°C 		v 				h 			u 		s 			cp 		Y 		L		n		s	
-20		1,006580	
0 		1,000160 		0,06 		-0,04 	-0,0001 	4,228 	-0,080 	561,0 	1792 	75,65
4		1,000028
5 		1,0000 		21,1 		21,0 	0,076 		4,200 	0,011 	570,6 	1518 	74,95
10 		1,0003 		42,1 		42,0 	0,151 		4,188 	0,087 	580,0 	1306 	74,22
15 		1,0009 		63,0 		62,9 	0,224 		4,184 	0,152 	589,4 	1137 	73,49
20 		1,001797 		83,9 		83,8 	0,296 		4,183 	0,209 	598,4 	1001 	72,74
25 		1,0029 		104,8 		104,7 	0,367 		4,183 	0,259 	607,2 	890,4 	71,98
30 		1,0044 		125,8 		125,7 	0,437 		4,183 	0,305 	615,5 	797,7 	71,20
35 		1,0060 		146,7 		146,6 	0,505 		4,183 	0,347 	623,3 	719,6 	70,41
40 		1,007842 		167,58 	167,5 	0,572 		4,182 	0,386 	630,6 	653,3 	69,60
45 		1,0099 		188,5 		188,4 	0,638 		4,182 	0,423 	637,3 	596,3 	68,78
50 		1,0121 		209,4 		209,3 	0,704 		4,181 	0,457 	643,6 	547,1 	67,95
60 		1,017089 		251,2 		251,1 	0,831 		4,183 	0,522 	654,4 	466,6 	66,24
70 		1,0227 		293,1 		293,0 	0,955 		4,187 	0,583 	663,1 	404,1 	64,49
80 		1,029027 		335,0 		334,9 	1,075 		4,194 	0,640 	670,0 	354,5 	62,68
90 		1,0359 		377,0 		376,9 	1,193 		4,204 	0,696 	675,3 	314,6 	60,82
99,63 	1,0431 		417,5 		417,4 	1,303 		4,217 	0,748 	679,0 	283,0 	58,99
100	1,043453		419,1

Stoffdaten von Wasser Quelle Wickipedia

Wasser hat unter Normaldruck seine größte Dichte von 1000 Kilogramm pro Kubikmeter bei 3,98 °C und zeigt damit eine Dichteanomalie. 
Diese besteht darin, dass sich Wasser unterhalb von 3,98 °C bei weiterer Temperaturverringerung, auch beim Wechsel zum festen 
Aggregatzustand, wieder ausdehnt, was man nur von wenigen Stoffen kennt. Die derzeit genauesten publizierten Werte für die maximale 
Dichte liegen bei (999,974950 ± 0,00084) kg/m³ und bei (3,983 ± 0,00067) °C für die Temperatur, bei der dieser Wert erreicht wird. 
Die Werte stellen einen Mittelwert der von verschiedenen physikalischen Instituten veröffentlichten Zahlen dar (Stand 2001).

Die Berechnung der Dichte von luftfreiem Wasser DLF in Abhängigkeit von der Temperatur T ([T] = °C) kann mit Hilfe der folgenden 
Virialgleichung erfolgen:
: \frac{D_{\rm LF}}{\rm g/l} = \frac{a_0 + a_1 T + a_2 T^2 + a_3 T^3 + a_4 T^4 + a_5 T^5}{1 + b T}.
mit den Koeffizienten: a0 = 999,83952; a1 = 16,952577 (°C)-1; a2 = -7,9905127·10-3 (°C)-2; a3 = -4,6241757·10-5 (°C)-3; 
a4 = 1,0584601·10-7 (°C)-4; a5 = -2,8103006·10-10 (°C)-5 und b = 0,0168872. 
Für die Berechnung der Dichte von luftgesättigtem Wasser korrigiert man den Wert nach 
DLG/(g/l) = DLF/(g/l) - 0,004612 + 0,000106 (°C)-1·T. (Quelle: PTB-Mitteilungen 100/3-90)

*)
END_FUNCTION

(* POU Mathematical/functions/LINEAR_INT, ST *)
FUNCTION LINEAR_INT : REAL
VAR_INPUT
	X : REAL;
	XY : ARRAY[1..20,0..1] OF REAL;
	Pts : INT;
END_VAR
VAR
	i : INT;
END_VAR

(*
	version 1.1	27 dec 2007
	programmer 	oscat
	tested BY		oscat

LINEAR_INT calculates an output based on a linear interpolation of up to 20 coordinates given in an array
the input coordinates have to start at the lowest array position and must be sorted ba ascending X values.

*)
(*make sure n is bound within the array size *)
pts := MIN(pts,20);

(* calculate the linear segement interpolation *)
i := 2;
(* search for segment and calculate output
	below and above the defined segments we interpolate the last segment *)
WHILE (i < pts) AND (XY[i,0] < X) DO
	i := i + 1;
END_WHILE;

(* calculate the output value on the corresponding segment coordinates *)
LINEAR_INT := ((XY[i,1] - XY[i-1,1]) * X - XY[i,1] * XY[i-1,0] + XY[i-1,1] * XY[i,0]) / (XY[i,0] - XY[i-1,0]);

(* revision history
hm	7. oct 2007		rev 1.0
	original version

hm	27 dec 2007		rev 1.1
	changed code for better performance
*)
END_FUNCTION

(* POU Building/HLK/Heat_temp, ST *)
FUNCTION_BLOCK Heat_temp
VAR_INPUT
	T_ext : REAL;
	Offset : REAL;
	t_req : REAL;
END_VAR
VAR_INPUT CONSTANT
	TY_max : REAL := 70;
	TY_min : REAL := 20;
	T_int : REAL := 20;
	TY_config : REAL := 50;
	T_ext_config : REAL := -15;
	C : REAL := 1.33;
END_VAR
VAR_OUTPUT
	Ty : REAL;
END_VAR
VAR
END_VAR

(*
version 1.0	27 jan 2007
programmer 	hugo
tested by		tobias

Heat_Temp calculates a heat characteristic based on the formula: tv=ti+(tvmax-ti)*((ti-tau)/(ti-taumin))^(1/n)
while
tv necessary heating temperature.
ti internal room temperature (20°C)
tau current external temperature
external temperature to determine characteristics
C exponent for heating system (normally 1,33 or 1,1 for floor heating)

The two additional inputs TY_min and TY_max set limits for the output TY, while an offset inputs allows to rise or lower the room temperature.

*)
IF t_ext > t_int + Offset THEN
	ty := t_int + offset;
ELSE
Ty := T_int - offset + (TY_config - T_int) * EXPT((T_int - offset - T_ext) / (T_int - offset - T_ext_config),1 / C);
END_IF;
IF t_req > ty THEN ty := t_req; END_IF;
ty := LIMIT(TY_min, ty, TY_max);



(*

tv=ti+(tvmax-ti)*((ti-tau)/(ti-taumin))^(1/n)

tv aktuelle Vorlauftemp.
ti Raumtemperatur innen (20°C)
tau aktuelle Außentemperatur
taumin minimale Außentemperatur -12°C oder -15°C
n Heizkörperexponent (meistens 1,33)
Fußbodenheizung = 1,1
Wandheizung 1,3

Normen z. B. DIN 4703, DIN 4725 oder die Literatur, z. B Recknagel Abschnitt 1.3.5.

*)
END_FUNCTION_BLOCK

(* POU Building/HLK/legionella, ST *)
FUNCTION_BLOCK legionella
VAR_INPUT
	manual : BOOL;
	temp_boiler : REAL;
	temp_return : REAL := 100;
	DT_in: DT;
	rst : BOOL;
END_VAR
VAR_INPUT CONSTANT
	T_start: TOD := tod#03:00:00;
	day : INT := 7;
	temp_set : REAL := 70;
	temp_offset : REAL := 10;
	temp_hys : REAL := 5;
	t_max_heat: TIME := t#10m;
	t_max_ret : TIME := t#10m;
	tp_0: TIME := t#5m;
	tp_1: TIME := t#5m;
	tp_2: TIME := t#5m;
	tp_3: TIME := t#5m;
	tp_4: TIME := t#5m;
	tp_5: TIME := t#5m;
	tp_6: TIME := t#5m;
	tp_7: TIME := t#5m;
END_VAR
VAR_OUTPUT
	Heat : BOOL;
	pump : BOOL;
	valve0 : BOOL;
	valve1 : BOOL;
	valve2 : BOOL;
	valve3 : BOOL;
	valve4 : BOOL;
	valve5 : BOOL;
	valve6 : BOOL;
	valve7 : BOOL;
	run: BOOL;
	Status : BYTE;
END_VAR
VAR
	X1: timer_1;
	x2: sequence_8;
	x3: hyst_1;
	init: BOOL;
END_VAR

(*
version 1.1	17. jan 2007
programmer 	oscat
tested by		hans

Legionella is a complete sequencer for up to 8 hot water lines that need to be sterilzed periodically.
legionella needs a DT input with the appropriate time, usually gererated by the rtc of the system. for system independence this time is connected externally.
T_start is the time when sterilazation should be started and day is the day_of_week when it should be performed (1=Monday and 7=sunday).
so sterilazation is autioimatically performed once a week at a specified time.
temp_set and temp_hys and temp_offset specify the boiler temperatur nedded for sterilization. as a defaut Temp_set is set to 70 deg C and Temp_hys is set to 5 deg C and temp_offset is 10 deg C.
a temp boiler input reads the boiler temperature of the hot water tank.
after a start pulse is gererated by the weekly timer or a manual test input the sequence is started:
1. the boiler is heated to temp_set + temp_offset + temp_hys = 85 deg C unless chaged at setup.
	the heat output is turned on and tells the heater to turn heating on. if the temp is not reached for a time of t_max_heat (10 min) the error output is set and the sequence is stopped.
2. after the specified temperature is reached, the output valve0 and pump is turned on and starts sterilization of line0 until temp_return has reached temp_set and continues to sterilize for a time of tp_0 (5 min default).
	if tmep_set is not reached at the temp_return_input then the error output is set and the sequence will be stopped.
	if there is no temp sensor for temp_return (the temperature at the return point for the circulation pump pls set this imput to a value greater then temp_set (by default use 100 deg C).
	in this case sterilization is performed for the default times without monitoring the return temp.
3. this sequence is repeated for up to valves.

connection scheme:

temp_boiler:	input oif the boiler temperature sensor.
temp_hys:		config value for the heater hysteresis, preset to 5 deg C.
temp_offset:	config value for the heater temp_offset against temp_set, preset to 10 deg C.
temp_set:		config value for the specified sterilization temperature, preset to 70 deg C.
temp_return:	input of the circulation return line temperature sensor, if not availabe set this value to 100 deg C.
manual:		manual input to start the sterilization by hand for diagnostic purposes, rising edge active, leave low for automatic operation.
DT_in:			date,time input supplied by a external real time clock.
T_start:		time of day when the sterilization should be started.
day:			config value for day of week when the process should be started, preset to sunday.
t_max_hest:	tmax time to be needed for the heater to heat the hot water tank to the specified value, preset to 10 min.

*)
(* startup initialization *)
IF NOT init THEN
	init := TRUE;
	X1.start_day := day;
	X1.start_time := T_start;
	X3.low := Temp_offset + temp_set;
	X3.high := Temp_hys + X3.low;
	X2.wait0 := T_max_heat;
	X2.delay0 := TP_0;
	X2.delay1 := TP_1;
	X2.delay2 := TP_2;
	X2.delay3 := TP_3;
	X2.delay4 := TP_4;
	X2.delay5 := TP_5;
	X2.delay6 := TP_6;
	X2.delay7 := TP_7;
	X2.wait1 := T_max_ret;
	X2.wait2 := T_max_ret;
	X2.wait3 := T_max_ret;
	X2.wait4 := T_max_ret;
	X2.wait5 := T_max_ret;
	X2.wait6 := T_max_ret;
	X2.wait7 := T_max_ret;
	X2();
END_IF;

(* oerational code *)
X1(DT_in := DT_in);
IF X1.Q OR manual OR x2.run THEN
	X3(in := temp_boiler);
	X2.in0 := X3.Q OR x3.win;
	X2.in1 := temp_return >= temp_set;
	X2.in2 := x2.in1;
	X2.in3 := x2.in1;
	X2.in4 := x2.in1;
	X2.in5 := x2.in1;
	X2.in6 := x2.in1;
	X2.in7 := x2.in1;
	X2.rst := rst;
	X2(start := X1.Q OR manual);
	run := x2.run;
	pump := x2.any;
	Heat := NOT X3.Q AND x2.run;
	valve0 := X2.Q0;
	valve1 := X2.Q1;
	valve2 := X2.Q2;
	valve3 := X2.Q3;
	valve4 := X2.Q4;
	valve5 := X2.Q5;
	valve6 := X2.Q6;
	valve7 := X2.Q7;
	pump := X2.any;
	status := X2.status;
ELSE;
	X2(start :=0);
	status := x2.status;
END_IF;

(* revision history

hm 17.jan 2007	rev 1.1
	rewritten to st for higher performance
	changes eeror output to esr compatible status output
*)
END_FUNCTION_BLOCK

(* POU Logic/generators/sequence_8, ST *)
FUNCTION_BLOCK sequence_8
VAR_INPUT
	in0 : BOOL := TRUE;
	in1 : BOOL := TRUE;
	in2 : BOOL := TRUE;
	in3 : BOOL := TRUE;
	in4 : BOOL := TRUE;
	in5 : BOOL := TRUE;
	in6 : BOOL := TRUE;
	in7 : BOOL := TRUE;
	start : BOOL;
	rst : BOOL;
	wait0 : TIME := t#0s;
	delay0 : TIME := t#0s;
	wait1 : TIME := t#0s;
	delay1 : TIME := t#0s;
	wait2 : TIME := t#0s;
	delay2 : TIME := t#0s;
	wait3 : TIME := t#0s;
	delay3 : TIME := t#0s;
	wait4 : TIME := t#0s;
	delay4 : TIME := t#0s;
	wait5 : TIME := t#0s;
	delay5 : TIME := t#0s;
	wait6 : TIME := t#0s;
	delay6 : TIME := t#0s;
	wait7 : TIME := t#0s;
	delay7 : TIME := t#0s;
END_VAR
VAR_INPUT CONSTANT
	stop_on_error : BOOL := FALSE;
END_VAR
VAR_OUTPUT
	Q0 : BOOL;
	Q1 : BOOL;
	Q2 : BOOL;
	Q3 : BOOL;
	Q4 : BOOL;
	Q5 : BOOL;
	Q6 : BOOL;
	Q7 : BOOL;
	any : BOOL;
	run: BOOL;
	step : INT := -1;
	status : BYTE;
END_VAR
VAR
	last : TIME;
	edge : BOOL;
	tx: TIME;
	init: BOOL;
END_VAR

(*
version 1.4	17 sep 2007
programmer 	oscat
tested by		hans

sequence_8 enables run when a low to high transition is present on start.
a low to high transition on start will restart the sequencer at any time while a rst will hold the sequencer in reset while true.
after run is enabled with a rising edge on start the sequencer waits for wait0 on in0 to enable q0 which stays on for delay0.
the next cycle starts with wait1, continues with delay 1 and so on...
if an edge is not detected during the wait period, the sequencer will then display the error number on the status output.
The status numbers are 1 .. 8 for erros in step 0..7.
after the last step that sets q7, the sequencer leaves q7 on for delay7 and then resets to the initial state.
a step output will indicate the current step of the sequencer and will also be present with a fault condition.
after the first output is turened on the sequencer switches from q0 to q1 and so on, at any time there is only one output enabled.
if an input signal is not detected during a wait period, the sequencer will display the error number ( 1 for in0, 2 for in1 .... ).
when an error is present and the config variable stop_on_error is set then the sequencer will stop. otherwise it will continue.
The status output will also display 110 for waiting and 111 sequece running.

*)
(* read sps timer *)
tx := DWORD_TO_TIME(T_PLC_MS());

(* initialize on startup *)
IF NOT init THEN
	last := tx;
	init := TRUE;
	status := 110;
END_IF;

(* asynchronous reset *)
IF rst THEN
	step := -1;
	Q0 := 0;
	Q1 := 0;
	Q2 := 0;
	Q3 := 0;
	Q4 := 0;
	Q5 := 0;
	Q6 := 0;
	Q7 := 0;
	status := 110;
	run := 0;

(* edge on start input restarts the sequencer *)
ELSIF start AND NOT edge THEN
	step := 0;
	last := tx;
	status := 111;
	Q0 := 0;
	Q1 := 0;
	Q2 := 0;
	Q3 := 0;
	Q4 := 0;
	Q5 := 0;
	Q6 := 0;
	Q7 := 0;
	run := 1;
END_IF;
edge := start;

(* check if stop on error is necessary *)
IF status > 0 AND status < 100 AND stop_on_error THEN RETURN; END_IF;

(* sequence is running *)
IF run AND step = 0 THEN
	IF NOT q0 AND in0 AND tx - last <= wait0 THEN
		Q0 := TRUE;
		last := tx;
	ELSIF NOT q0 AND tx - last > wait0 THEN
		status := 1;
		run := FALSE;
	ELSIF q0 AND tx - last >= delay0 THEN
		step := 1;
		last := tx;
	END_IF;
END_IF;
IF run AND step = 1 THEN
	IF NOT q1 AND in1 AND tx - last <= wait1 THEN
		Q0 := FALSE;
		Q1 := TRUE;
		last := tx;
	ELSIF NOT q1 AND Tx - last > wait1 THEN
		status := 2;
		q0 := FALSE;
		run := FALSE;
	ELSIF q1 AND tx - last >= delay1 THEN
		step := 2;
		last := tx;
	END_IF;
END_IF;
IF run AND step = 2 THEN
	IF NOT q2 AND in2 AND tx - last <= wait2 THEN
		Q1 := FALSE;
		Q2 := TRUE;
		last := tx;
	ELSIF NOT q2 AND Tx - last > wait2 THEN
		status := 3;
		q1 := FALSE;
		run := FALSE;
	ELSIF q2 AND tx - last >= delay2 THEN
		step := 3;
		last := tx;
	END_IF;
END_IF;
IF run AND step = 3 THEN
	IF NOT q3 AND in3 AND tx - last <= wait3 THEN
		Q2 := FALSE;
		Q3 := TRUE;
		last := tx;
	ELSIF NOT q3 AND Tx - last > wait3 THEN
		status := 4;
		q2 := FALSE;
		run := FALSE;
	ELSIF q3 AND tx - last >= delay3 THEN
		step := 4;
		last := tx;
	END_IF;
END_IF;
IF run AND step = 4 THEN
	IF NOT q4 AND in4 AND tx - last <= wait4 THEN
		Q3 := FALSE;
		Q4 := TRUE;
		last := tx;
	ELSIF NOT q4 AND Tx - last > wait4 THEN
		status := 5;
		q3 := FALSE;
		run := FALSE;
	ELSIF q4 AND tx - last >= delay4 THEN
		step := 5;
		last := tx;
	END_IF;
END_IF;
IF run AND step = 5 THEN
	IF NOT q5 AND in5 AND tx - last <= wait5 THEN
		Q4 := FALSE;
		Q5 := TRUE;
		last := tx;
	ELSIF NOT q5 AND Tx - last > wait5 THEN
		status := 6;
		q4 := FALSE;
		run := FALSE;
	ELSIF q5 AND tx - last >= delay5 THEN
		step := 6;
		last := tx;
	END_IF;
END_IF;
IF run AND step = 6 THEN
	IF NOT q6 AND in6 AND tx - last <= wait6 THEN
		Q5 := FALSE;
		Q6 := TRUE;
		last := tx;
	ELSIF NOT q6 AND Tx - last > wait6 THEN
		status := 7;
		q5 := FALSE;
		run := FALSE;
	ELSIF q6 AND tx - last >= delay6 THEN
		step := 7;
		last := tx;
	END_IF;
END_IF;
IF run AND step = 7 THEN
	IF NOT q7 AND in7 AND tx - last <= wait7 THEN
		Q6 := FALSE;
		Q7 := TRUE;
		last := tx;
	ELSIF NOT q7 AND Tx - last > wait7 THEN
		status := 8;
		q6 := FALSE;
		run := FALSE;
	ELSIF q7 AND tx - last >= delay7 THEN
		step := -1;
		Q7 := FALSE;
		Run := FALSE;
		status := 110;
	END_IF;
END_IF;
any := q0 OR q1 OR q2 OR q3 OR q4 OR q5 OR q6 OR q7;

(*
hm 1.10.06		rev 1.1
	corrected delay logic to be after event and not before
	added any output

hm 1.12.06		rev 1.2
	corrected failure in sequence logic.
	added init at startup to prevent from initial statuss after start.

hm 17.1.2007		rev 1.3
	changed output fault to status for better compatibility with other modules (ESR)
	added stop on error functionality and setup variable
	default for inputs in0..7 is true.
	renames variable state to step

hm	17.sep 2007		rev 1.4
	replaced time() with T_PLC_MS() for compatibility reasons

*)
END_FUNCTION_BLOCK

(* POU Engineering/control/hyst_1, ST *)
FUNCTION_BLOCK hyst_1
VAR_INPUT
	In : REAL;
	high : REAL;
	low : REAL;
END_VAR
VAR_OUTPUT
	Q : BOOL := 0;
	win : BOOL := 0;
END_VAR
VAR
END_VAR

(*
	version 1.0	4 aug 2006
	programmer 	hugo
	tested BY		tobias

this hysteresis function switches the output high if the input signal reaches obove high and will switch to low when the input falls back below low value.
a separate output mid is set if the input stays between low and high value.

*)
IF Q THEN
	IF in < low THEN q := FALSE; END_IF;
ELSE
	IF in > high THEN q := TRUE; END_IF;
END_IF;
win := in > low AND in < high;
END_FUNCTION_BLOCK

(* POU Building/HLK/temp_ext, ST *)
FUNCTION_BLOCK temp_ext
VAR_INPUT
	t_ext1 : REAL;
	t_ext2 : REAL;
	t_ext3 : REAL;
	t_ext_config : BYTE := 0;
	dt_in : DT;
END_VAR
VAR_INPUT CONSTANT
	t_ext_min : REAL := -40;
	t_ext_max : REAL := 60;
	t_ext_default : REAL := -10;
	heat_period_start : DATE := D#1970-9-1;
	heat_period_stop : DATE := D#1970-4-30;
	cool_period_start : DATE := D#1970-4-1;
	cool_period_stop : DATE := D#1970-9-30;
	heat_start_temp_day : REAL := 15;
	heat_start_temp_night : REAL := 10;
	heat_stop_temp : REAL := 18;
	cool_start_temp_day : REAL := 26;
	cool_start_temp_night : REAL := 26;
	cool_stop_temp : REAL := 24;
	start_day : TOD := tod#09:00;
	start_night : TOD := tod#21:00;
	cycle_time : TIME := t#10m;
END_VAR
VAR_OUTPUT
	t_ext : REAL;
	heat : BOOL;
	cool : BOOL;
END_VAR
VAR
	tx: TIME;
	last_run: TIME;
	init: BOOL;
	cool_start: DATE;
	cool_stop: DATE;
	heat_start: DATE;
	heat_stop: DATE;
	xdate: DATE;
	day: BOOL;
END_VAR


(*
version 1.1	15 sep 2007
programmer 	hugo
tested by		tobias

temp_ext measures and processes ext temperature and decides if heating or cooling is needed.

 the measurement of t_ext has 3 inputs which can be configured in different ways:
	t_ext_config = 0 means the ext temp is the avg of the 3 external temperatures, this mode is the default mode.
	t_ext_config = 1 means t_ext1 is used.
	t_ext_config = 2 means t_ext1 is used.
	t_ext_config = 3 means t_ext1 is used.
	t_ext_config = 4 means t_ext_default is used.
	t_ext_config = 5 means the lowest of the 3 external temperatures is used.
	t_ext_config = 6 means the higest externnal temperature is used.
	t_ext_config = 7 means the midlle external temperature is used, if there are only two working, the lowest is used.
	in any config mode, an external temperature higher then t_ext_max or lower then t_ext_min is ignored to prevent from temperatures caused by broken sensors or wires.
	if no external temperature is available, a default value (t_ext_default) is used.
	if you have only one external sensor, connect the 3 inputs to the same sensor, or select the right input with t_ext_config.

heating or cooling is enabled during heating / cooling period when the day or night start temperature is reached for at least the specified delay time and will be disabled after the stop temperature is reached. 
t_ext output can be used by other modules to determine the correct system temperature for heating or cooling.

*)
IF NOT init THEN
	init := TRUE;
	heat_start := set_Date(1972,month(heat_period_start),day_of_month(heat_period_start));
	heat_stop := set_Date(1972,month(heat_period_stop),day_of_month(heat_period_stop));
	cool_start := set_Date(1972,month(cool_period_start),day_of_month(cool_period_start));
	cool_stop := set_Date(1972,month(cool_period_stop),day_of_month(cool_period_stop));
END_IF;

(* read system time *)
tx := DWORD_TO_TIME(T_PLC_MS());

(* for efficiency exit isf this program has been executed less then 1min ago *)
IF tx - last_run < cycle_time THEN RETURN; END_IF;

(* calculate frequently used variables *)
xdate := set_Date(1972,month(DT_TO_DATE(dt_in)),day_of_month(DT_TO_DATE(dt_in)));
day := DT_TO_TOD(dt_in) >= start_day AND  DT_TO_TOD(dt_in) < start_night;

(* read the correct external temperature depending on the t_ext_config setting *)
t_ext := multi_in(t_ext1, t_ext2, t_ext3, t_ext_default, t_ext_min, t_ext_max, t_ext_config);

(* dtermine heating *)
IF (heat_start <= heat_stop AND xdate >= heat_start AND xdate <= heat_stop) OR (heat_start > heat_stop AND (xdate >= heat_start OR xdate <= heat_stop)) THEN
	(* heating period id true check for temperature *)
	IF day AND t_ext <= heat_start_temp_day THEN
		heat := TRUE;
	ELSIF NOT day AND t_ext <= heat_start_temp_night THEN
		heat := TRUE;
	ELSIF t_ext >= heat_stop_temp THEN
		heat := FALSE;
	END_IF;
ELSE
	heat := FALSE;
END_IF;

(* dtermine cooling *)
IF (cool_start <= cool_stop AND xdate >= cool_start AND xdate <= cool_stop) OR (cool_start > cool_stop AND (xdate >= cool_start OR xdate <= cool_stop)) THEN
	(* cooling period is true check for temperature *)
	IF day AND t_ext >= cool_start_temp_day THEN
		cool := TRUE;
	ELSIF NOT day AND t_ext >= cool_start_temp_night THEN
		cool := TRUE;
	ELSIF t_ext <= cool_stop_temp THEN
		cool := FALSE;
	END_IF;
ELSE
	cool := FALSE;
END_IF;

last_run := tx;

(* revision history
hm	6 dec 2006		rev 1.0
	original version

hm	15.9.2007		rev 1.1
	replaced Time() with T_PLC_MS for compatibility and performance reasons

*)
END_FUNCTION_BLOCK

(* POU Engineering/sensor/multi_in, ST *)
FUNCTION multi_in : REAL
VAR_INPUT
	in_1 : REAL;
	in_2 : REAL;
	in_3 : REAL;
	default : REAL;
	in_min : REAL;
	in_max : REAL;
	mode : BYTE;
END_VAR
VAR
	count: INT;
	F1: BOOL;
	F2: BOOL;
	F3: BOOL;
END_VAR

(*

version 1.1	1 jan 2007
programmer 	oscat
tested by		hugo

multi_in is a signal conditioning function ehich can be configured in 8 different ways.
it is used to read multiple sensors for the same value and protect the user from broken sensors or invalid data from sensors.

multi_in can be configured in different ways:
	mode = 0 means the the avg of the 3 inputs is used, this mode is the default mode.
	mode = 1 means in_1 is used.
	mode = 2 means in_2 is used.
	mode = 3 means in_3 is used.
	mode = 4 means default is used.
	mode = 5 means the lowest of the 3 external temperatures is used.
	mode = 6 means the higest externnal temperature is used.
	mode = 7 means the midlle input is used, if there are only two working, the lowest input is used.
	mode > 7 ,eans output is 0 at all times.
	in any config mode, an input higher then in_max or lower then in_min is ignored to prevent values from broken sensors or wires.
	if all inputs are higher then in_max or lower then in_min, a default value (default) is used.
*)
IF  in_1 > in_min AND in_1 < in_max THEN F1 := TRUE; ELSE F1 := FALSE; END_IF;
IF  in_2 > in_min AND in_2 < in_max THEN F2 := TRUE; ELSE F2 := FALSE; END_IF;
IF  in_2 > in_min AND in_3 < in_max THEN F3 := TRUE; ELSE F3 := FALSE; END_IF;

CASE mode OF
0:	count := 0;
	IF F1 THEN
		count := count + 1;
		multi_in := in_1;
	ELSE
		multi_in := 0;
	END_IF;
	IF F2 THEN
		count := count + 1;
		multi_in := multi_in + in_2;
	END_IF;
	IF F3 THEN
		count := count + 1;
		multi_in := multi_in + in_3;
	END_IF;
	IF count = 0 THEN
		multi_in := default;
	ELSE
		multi_in := multi_in / count;
	END_IF;

1:	IF F1 THEN multi_in := in_1; ELSE multi_in := default; END_IF;

2:	IF F2 THEN multi_in := in_2; ELSE multi_in := default; END_IF;

3:	IF F3 THEN multi_in := in_3; ELSE multi_in := default; END_IF;

4:	multi_in := default;

5:	IF F1 THEN multi_in := in_1; ELSE multi_in := in_max; END_IF;
	IF F2 AND in_2 < multi_in THEN multi_in := in_2; END_IF;
	IF F3 AND in_3 < multi_in THEN multi_in := in_3; END_IF;
	IF multi_in = in_max THEN multi_in := default; END_IF;

6:	IF F1 THEN multi_in := in_1; ELSE multi_in := in_min; END_IF;
	IF F2 AND in_2 > multi_in THEN multi_in := in_2; END_IF;
	IF F3 AND in_3 > multi_in THEN multi_in := in_3; END_IF;
	IF multi_in = in_min THEN multi_in := default; END_IF;

7:	IF F1 AND F2 AND F3 THEN multi_in := mid3(in_1, in_2, in_3);
	ELSIF F1 AND F2 THEN multi_in := MIN(in_1, in_2);
	ELSIF F1 AND F3 THEN multi_in := MIN(in_1, in_3);
	ELSIF F2 AND F3 THEN multi_in := MIN(in_2, in_3);
	ELSIF F1 THEN multi_in := in_1;
	ELSIF F2 THEN multi_in := in_2;
	ELSIF F3 THEN multi_in := in_3;
	ELSE multi_in := default;
	END_IF;

END_CASE;

(*
hm 1.1.2007	rev 1.1
	changed midr to mid3 function

*)
END_FUNCTION

(* POU Mathematical/MID3, ST *)
FUNCTION MID3 : REAL
VAR_INPUT
	in1 : REAL;
	in2 : REAL;
	in3 : REAL;
END_VAR
VAR
END_VAR

(*
version 1.1	1 jan 2007
programmer 	hugo
tested by		tobias

returns the mid value of 3 real inputs.

*)
IF (in1 <= in2) AND (in1 >= in3) OR (in1 >= in2) AND (in1 <= in3) THEN
	mid3 := in1;
ELSIF (in2 <= in1) AND (in2 >= in3) OR (in2 >= in1) AND (in2 <= in3) THEN
	mid3 := in2;
ELSE
	mid3 := in3;
END_IF;

(*
hm	1.1.2007	rev 1.1
	rewrote the function for better performance

*)
END_FUNCTION

(* POU Building/HLK/water_CP, ST *)
FUNCTION water_CP : REAL
VAR_INPUT
	T : REAL;
END_VAR
VAR
	Pts : INT := 10;
	data : ARRAY[1..20, 0..1] OF REAL := 0,4.228, 5,4.20, 10,4.188, 15,4.184, 50,4.181, 60,4.183, 70,4.187, 80,4.194, 90,4.204, 100,4.22;
END_VAR

(*
version 1.1	27 dec 2007 
programmer 	hugo
tested by	tobias

water_cp calculates the specific heat capacity of liquid water from 0..100 °C 

*)
water_CP := LINEAR_INT(T, Data, Pts);


(* revision history

hm	29.10.2007		rev 1.0
	original version

hm	27. dec 2007	rev 1.1
	increased accuracy

*)

(*
    °C - die Celsius-Temperatur in Grad Celsius
    v – das spezifische Volumen in Kubikdezimeter je Kilogramm dm³/kg
    h – die spezifische Enthalpie in Kilojoule je Kilogramm 	kJ/kg
    u – die spezifische Innere Energie in Kilojoule je Kilogramm 	kJ/kg
    s – die spezifische Entropie in Kilojoule je Kilogramm mal Kelvin 	kJ/(kg·K)
    cp - die spezifische Wärmekapazität bei konstantem Druck in Kilojoule je Kilogramm mal Kelvin 	kJ/(kg·K)
    Y – Volumenausdehnungskoeffizient in 10-3 durch Kelvin  10-3/K
    L – Wärmeleitfähigkeit in Milliwatt je Meter mal Kelvin  mW / (m·K) 
    n – Viskosität in Mikropascal mal Sekunde uPa·s 	
    s ? – Oberflächenspannung in Millinewton je Meter  mN/m


°C 		v 				h 			u 		s 			cp 		Y 		L		n		s	
-20		1,006580	
0 		1,000160 		0,06 		-0,04 	-0,0001 	4,228 	-0,080 	561,0 	1792 	75,65
4		1,000028
5 		1,0000 		21,1 		21,0 	0,076 		4,200 	0,011 	570,6 	1518 	74,95
10 		1,0003 		42,1 		42,0 	0,151 		4,188 	0,087 	580,0 	1306 	74,22
15 		1,0009 		63,0 		62,9 	0,224 		4,184 	0,152 	589,4 	1137 	73,49
20 		1,001797 		83,9 		83,8 	0,296 		4,183 	0,209 	598,4 	1001 	72,74
25 		1,0029 		104,8 		104,7 	0,367 		4,183 	0,259 	607,2 	890,4 	71,98
30 		1,0044 		125,8 		125,7 	0,437 		4,183 	0,305 	615,5 	797,7 	71,20
35 		1,0060 		146,7 		146,6 	0,505 		4,183 	0,347 	623,3 	719,6 	70,41
40 		1,007842 		167,58 	167,5 	0,572 		4,182 	0,386 	630,6 	653,3 	69,60
45 		1,0099 		188,5 		188,4 	0,638 		4,182 	0,423 	637,3 	596,3 	68,78
50 		1,0121 		209,4 		209,3 	0,704 		4,181 	0,457 	643,6 	547,1 	67,95
60 		1,017089 		251,2 		251,1 	0,831 		4,183 	0,522 	654,4 	466,6 	66,24
70 		1,0227 		293,1 		293,0 	0,955 		4,187 	0,583 	663,1 	404,1 	64,49
80 		1,029027 		335,0 		334,9 	1,075 		4,194 	0,640 	670,0 	354,5 	62,68
90 		1,0359 		377,0 		376,9 	1,193 		4,204 	0,696 	675,3 	314,6 	60,82
99,63 	1,0431 		417,5 		417,4 	1,303 		4,217 	0,748 	679,0 	283,0 	58,99
100	1,043453		419,1

Stoffdaten von Wasser Quelle Wickipedia

Wasser hat unter Normaldruck seine größte Dichte von 1000 Kilogramm pro Kubikmeter bei 3,98 °C und zeigt damit eine Dichteanomalie. 
Diese besteht darin, dass sich Wasser unterhalb von 3,98 °C bei weiterer Temperaturverringerung, auch beim Wechsel zum festen 
Aggregatzustand, wieder ausdehnt, was man nur von wenigen Stoffen kennt. Die derzeit genauesten publizierten Werte für die maximale 
Dichte liegen bei (999,974950 ± 0,00084) kg/m³ und bei (3,983 ± 0,00067) °C für die Temperatur, bei der dieser Wert erreicht wird. 
Die Werte stellen einen Mittelwert der von verschiedenen physikalischen Instituten veröffentlichten Zahlen dar (Stand 2001).

Die Berechnung der Dichte von luftfreiem Wasser DLF in Abhängigkeit von der Temperatur T ([T] = °C) kann mit Hilfe der folgenden 
Virialgleichung erfolgen:
: \frac{D_{\rm LF}}{\rm g/l} = \frac{a_0 + a_1 T + a_2 T^2 + a_3 T^3 + a_4 T^4 + a_5 T^5}{1 + b T}.
mit den Koeffizienten: a0 = 999,83952; a1 = 16,952577 (°C)-1; a2 = -7,9905127·10-3 (°C)-2; a3 = -4,6241757·10-5 (°C)-3; 
a4 = 1,0584601·10-7 (°C)-4; a5 = -2,8103006·10-10 (°C)-5 und b = 0,0168872. 
Für die Berechnung der Dichte von luftgesättigtem Wasser korrigiert man den Wert nach 
DLG/(g/l) = DLF/(g/l) - 0,004612 + 0,000106 (°C)-1·T. (Quelle: PTB-Mitteilungen 100/3-90)

*)
END_FUNCTION

(* POU Building/HLK/WCT, ST *)
FUNCTION WCT : REAL
VAR_INPUT
	T : REAL;
	V : REAL;
END_VAR
VAR
END_VAR

(*
version 1.1	7 dec 2007
programmer 	hugo
tested by		tobias

this function calculates the wind chill temperature

*)
IF V < 5 OR T > 10 THEN
	WCT := T;
ELSE
	WCT := 13.12 + 0.6215 * T +(0.3965 * T - 11.37) * EXP(LN(v) * 0.16);
END_IF;


(* revision history
hm		7 feb 2007
	original version

hm		7 dec 2007
	changed code for better performance

*)
END_FUNCTION

(* POU Building/Jalousie/blind_actuator, ST *)
 FUNCTION_BLOCK blind_actuator
VAR_INPUT
	UP, DN : BOOL;
	S_IN : BYTE;
	T_UD : TIME := T#10s;
	T_Angle : TIME := T#3s;
END_VAR
VAR_INPUT CONSTANT
	T_lockout : TIME := t#100ms;
END_VAR
VAR_OUTPUT
	pos, ang : BYTE;
	QU, QD : BOOL;
	status : BYTE;
END_VAR
VAR
	position, angle : rmp_B;
	lock : interlock;
END_VAR

(*
version 1.1	6 oct 2007
programmer 	hugo
tested by		tobias

blind actuator drives the up and down motor of a blind. T_lockout specifies the time between up or dn becomes active. 
To change direction there must be a minimum wait time to allow the motors to come to rest first.
the up and down outputs QU and QD are controlled by the inputs UP and DN.
the outputs pos and ang simulate the position of the blind pos = 0 means blind is down and pos = 255 = blind is up.
the angle 0 means vertical posisition of the slates and 255 means horizontal position of the slates.


*)
(* make sure only one motor is active at a given time *)
lock(i1 := UP, I2 := DN, TL := T_lockout);

(* ramp up or down to simulate the angle position of the blind slats *)
angle(en := lock.Q1 OR lock.Q2, UP := lock.Q1, PT := T_Angle);
position(en := lock.Q1 AND angle.high OR lock.Q2 AND angle.low, up := lock.Q1, PT := T_UD);

(* set the outputs *)
pos := position.Out;
ang := angle.Out;
QU := lock.Q1;
QD := lock.Q2;

(* set the status output *)
IF UP AND DN THEN
	IF s_in < 10 AND S_in > 1 THEN status := s_in; ELSE status := 1; END_IF;			(* error up and down together are not allowed *)
ELSIF S_IN > 0 THEN
	status := S_IN;
ELSIF UP THEN
	status := 101;
ELSIF DN THEN
	status := 102;
ELSE
	status := 0;
END_IF;


(* revision history
hm	29. sep 2007	rev 1.0
	original release

hm	6. oct 2007		rev 1.1
	rearranged outputs
	
*)
END_FUNCTION_BLOCK

(* POU Engineering/signal generators/rmp_B, ST *)
FUNCTION_BLOCK rmp_B
VAR_INPUT
	SET : BOOL := FALSE;
	PT : TIME;
	EN : BOOL := TRUE;
	UP : BOOL := TRUE;
	RST : BOOL := FALSE;
END_VAR
VAR_OUTPUT
	out : BYTE;
	busy: BOOL;
	high : BOOL;
	low : BOOL;
END_VAR
VAR
	last_step : DWORD;
	now : DWORD;
	tmp: DWORD;
	edge: BOOL;
	N : BYTE;
	init: BOOL;
END_VAR

(*
	version 1.6	25 dec 2007
	programmer 	oscat
	tested BY		oscat

this ramp generator generates a byte wide ramp with 255 steps
the generator has an asynchronous set and reset
the ramp is controlled by PT which is the total ramp time for a full sweep from 0..255
an UD input controlls the direction Up or Down and the E input enables the ramp generation
a busy output indicates that the ramp is running, busy false means output is stable.
the outputs low and high will be true when the output has reached its max or min value.

*)
(* read system time *)
now := T_PLC_MS();

(* init code for startup *)
IF NOT init THEN
	init := TRUE;
	last_step := now;
END_IF;

(* calculate the necessary step response *)
IF pt = t#0s THEN
	tmp := 255;
ELSE
	tmp := SHL(now - last_step, 8) / (TIME_TO_DWORD(pt));
END_IF;
IF tmp > 255 THEN N:= 255; ELSE N:= DWORD_TO_BYTE(tmp); END_IF;

(* detetct edge on en *)
IF en AND NOT edge THEN
	last_step := now;
(* check for asynchronous set or reset *)
ELSIF rst THEN
	out := 0;
ELSIF set  THEN
	out := 255;
ELSIF en AND N > 0 THEN
	(* generate ramp *)
	last_step := now;
	IF UP THEN
		IF out > 255 - N THEN out := 255; ELSE out := out + N; END_IF;
	ELSE
		IF out < N THEN out := 0; ELSE out := out - N; END_IF;
	END_IF;
END_IF;
edge := en;

(* checks for outputs stable and reset or set busy flag *)
IF out = 0 THEN
	busy := FALSE;
	low := TRUE;
	high := FALSE;
ELSIF out = 255 THEN
	busy := FALSE;
	high := TRUE;
	low := FALSE;
ELSE
	busy := en;
	high := FALSE;
	low := FALSE;
END_IF;


(* revision history

hm 5.10.2006	rev 1.1
	added busy output
hm 17.1.2007	rev 1.2
	renamed input ud to up for better usability
	deleted unused variable step

hm	17.9.2007	rev 1.3
	replaced time() with t_plc_ms() for compatibility reasons

hm	28. sep 2007	rev 1.4
	added outputs on and off
	busy is now disabled while en is false
	new coding for higher accuracy and performance

hm	5. oct 2007		rev 1.5
	added statements to allow for PT to be t#0s output jumps to max or min immediately

hm	25. dec 2007	REV 1.6
	IMPROOVED CODE FOR BETTER PERFORMANCE
*)
END_FUNCTION_BLOCK

(* POU Engineering/automation/interlock, ST *)
FUNCTION_BLOCK interlock
VAR_INPUT
	I1, I2 : BOOL;
	TL : TIME;
END_VAR
VAR_OUTPUT
	Q1, Q2 : BOOL;
END_VAR
VAR
	T1, T2 : TOF;
END_VAR

(*
version 1.0	28 sep 2007
programmer 	hugo
tested by		tobias

INTERLOCK has two inputs I1 and I2 which drive the corresponding outputs Q1 and Q2.
the inputs signals lock each other out and therfore I1 can only drive Q1 when I2 is Low and vice versa.
The input TL specifies a dead time between two outputs can become active.
an output can only become active when the other output was not active for the time TL.

*)
(* the input signal have a run delay to lockout the other input *)
T1(IN := I1, PT := TL);
T2(IN := I2, PT := TL);

Q1 := I1 AND NOT t2.Q;
Q2 := I2 AND NOT t1.Q;


(* revision history

hm	28 sep 2007		rev 1.0
	original version

*)
END_FUNCTION_BLOCK

(* POU Building/Jalousie/blind_control, ST *)
FUNCTION_BLOCK blind_control
VAR_INPUT
	UP, DN : BOOL;
	S_IN : BYTE;
	pi : BYTE;
	ai : BYTE;
	T_UD, T_ANGLE : TIME;
END_VAR
VAR_INPUT CONSTANT
	sens : BYTE := 5;
	T_Lockout: TIME := T#100ms;
END_VAR
VAR_OUTPUT
	pos, ang : BYTE;
	MU, MD : BOOL;
	status : BYTE;
END_VAR
VAR
	act : blind_actuator;
	delta : BYTE;
END_VAR

(*
version 1.3	30. oct 2007
programmer 	hugo
tested by		tobias


*)
IF UP AND DN THEN
	(* automatic modus detected *)
	(* first find correct position *)
	IF BYTE_TO_INT(act.pos) < BYTE_TO_INT(pi) - delta THEN
		act.UP := TRUE;
		act.DN := FALSE;
		delta := 0;
		act.S_IN := 121;
	ELSIF BYTE_TO_INT(act.pos) > BYTE_TO_INT(pi) + delta THEN
		act.UP := FALSE;
		act.DN := TRUE;
		delta := 0;
		act.S_IN := 122;
	(* regulate angle *)
	ELSIF BYTE_TO_INT(act.ang) < BYTE_TO_INT(ai) - delta AND T_angle > T#100ms THEN
		act.UP := TRUE;
		act.DN := FALSE;
		delta := 0;
		act.S_IN := 123;
	ELSIF BYTE_TO_INT(act.ang) > BYTE_TO_INT(ai) + delta AND T_angle > T#100ms THEN
		act.UP := FALSE;
		act.DN := TRUE;
		delta := 0;
		act.S_IN := 124;
	(* correct position reached *)
	ELSE
		act.UP := FALSE;
		act.DN := FALSE;
		delta := sens;
		act.S_IN := 0;
	END_IF;
ELSE
	act.UP := UP;
	act.DN := DN;
END_IF;

(* hand over status *)
IF s_in > 0 THEN act.S_IN := S_IN; END_IF;

(* blind control calls blind_actuator *)
act(T_UD:=T_UD, T_ANGLE:=T_ANGLE, T_lockout := T_Lockout);
pos := act.pos;
ang := act.ang;
MU := act.QU;
md := act.QD;
status := act.status;

(* revision history
hm	29. sep 2007	rev 1.0
	original release

hm	6. oct 2007		rev 1.1
	rearranged outputs
	integrated blind_actuator into blind_control

hm	16. oct 2007	rev 1.2
	ignore angle when t_angle = 0

hm 29. oct 2007	rev 1.3
	added lockout configuration time for motor direction change
	sens has a setup value of 5
*)
END_FUNCTION_BLOCK

(* POU Building/Jalousie/blind_input, ST *)
FUNCTION_BLOCK blind_input
VAR_INPUT
	pos, ang : BYTE;
	S1, S2 : BOOL;
	in : BOOL;
	pi, ai : BYTE;
END_VAR
VAR_INPUT CONSTANT
	single_switch : BOOL := FALSE;
	click_mode : BOOL := TRUE;
	click_time : TIME := T#200ms;
	click_timeout : TIME := T#60s;
	manual_timeout: TIME := T#1h;
END_VAR
VAR_OUTPUT
	QU, QD : BOOL;
	status : BYTE;
	po, ao : BYTE;
END_VAR
VAR
	click_run : TOF;
	tog1, tog2 : TOGGLE;
	pl1, pl2 : Pulse_Length;
	SU, SD : BOOL;
	last_act: DWORD;
	tx: DWORD;
END_VAR

(*
version 1.2	30 dec 2007
programmer 	hugo
tested by		tobias


*)
(* read system_time *)
tx := T_PLC_MS();

(* single or double switch operation *)
IF click_mode THEN
	PL1(in := S1, T_short := click_time, T_long := click_time);
	PL2(in := S2, T_short := click_time, T_long := click_time);
	(* a timeout needs to be added for click enable *)
	click_run(IN := pl1.short OR pl2.short, PT := click_timeout);
	tog1(clk := pl1.short, rst := pl1.long OR pl2.short OR pl2.long OR NOT click_run.Q);
	tog2(clk := pl2.short, rst := pl2.long OR pl1.short OR pl1.long OR NOT click_run.Q);

	SU := tog1.Q OR PL1.long;
	SD := tog2.Q OR pl2.long;
ELSE
	tog1(CLK := NOT S1);
	SU := (S1 AND NOT tog1.Q AND single_switch) OR (NOT single_switch AND S1);
	SD := (S1 AND tog1.Q AND single_switch) OR (NOT single_switch AND S2);
END_IF;

(* Forced Input is active *)
IF in THEN
	QU := TRUE;
	QD := TRUE;
	po := pi;
	ao := ai;
	status := 131;

(* in manual mode set ps and as to actual values *)
ELSIF SU OR SD THEN
	po := pos;
	ao := ang;
	last_act := tx;
	QU := SU;
	QD := SD;
	IF su THEN status := 132; ELSE status := 133; END_IF;

(* enable automatik mode after auto timer has expired *)
ELSIF manual_timeout > t#0s AND tx - last_act >= TIME_TO_DWORD(manual_timeout) THEN
	QU := TRUE;
	QD := TRUE;
	status := 134;

(* no input active *)
ELSE
	QU := FALSE;
	QD := FALSE;
	status := 0;
END_IF;


(* revision history
hm	29. sep 2007	rev 1.0
	original release

hm	6. oct 2007		rev 1.1
	renamed ps and as to po and ao

hm	30. dec 2007	rev 1.2
	added click_timeout variable and function

*)
END_FUNCTION_BLOCK

(* POU Logic/FF edge triggered/TOGGLE, ST *)
FUNCTION_BLOCK TOGGLE
VAR_INPUT
	CLK : BOOL;
	rst : BOOL := FALSE;
END_VAR
VAR_OUTPUT
	Q : BOOL;
END_VAR
VAR
	edge : BOOL;
END_VAR

(*
version 1.0	13 sep 2007
programmer 	hugo
tested by		tobias

toggle flip flop the output changes state with every rising edge of clk.

*)
IF rst THEN
	q := 0;
ELSIF clk AND NOT edge THEN
	Q := NOT Q;
END_IF;
edge := clk;

(* revision history

hm	13.9.2007		rev 1.0
	original version

*)
END_FUNCTION_BLOCK

(* POU Building/Jalousie/blind_night, ST *)
FUNCTION_BLOCK blind_night
VAR_INPUT
	UP, DN : BOOL;
	S_IN : BYTE;
	pi, ai : BYTE;
	E_night : BOOL := TRUE;
	E_day	: BOOL := TRUE;
	dtin : DT;
	sunrise, sunset : TOD;
END_VAR
VAR_INPUT CONSTANT
	sunrise_offset : TIME;
	sunset_offset : TIME;
	night_position : BYTE := 0;
	night_angle : BYTE := 0;
END_VAR
VAR_OUTPUT
	QU, QD : BOOL;
	status : BYTE;
	po, ao : BYTE;
END_VAR
VAR
	night : BOOL;
	last_night, last_day : DATE;
END_VAR

(*
version 1.2	6 oct 2007
programmer 	hugo
tested by		tobias


*)
IF NOT (up AND dn) AND night THEN
	(* manual operation at night will cancel operation for one night *)
	night := FALSE;
ELSIF (DT_TO_TOD(dtin) > sunset + sunset_offset) AND (last_night < DT_TO_DATE(dtin)) AND NOT night AND e_night THEN
	(* enable night *)
	night := TRUE;
	last_night := DT_TO_DATE(dtin);
ELSIF (DT_TO_TOD(dtin) > sunrise + sunrise_offset) AND (last_day < DT_TO_DATE(dtin)) AND night AND e_day AND (last_night < DT_TO_DATE(dtin)) THEN
	(* disable night *)
	night := FALSE;
	last_day := DT_TO_DATE(dtin);
END_IF;

(* shade at night only in auto mode and enable = true *)
IF UP AND DN AND night THEN
	status := 141;
	po := night_position;
	ao := night_angle;
ELSE
	QU := UP;
	QD := DN;
	po := pi;
	ao := ai;
	status := s_in;
END_IF;


(* revision history
hm	29. sep 2007	rev 1.0
	original version

hm	5. oct 2007		rev 1.1
	added enable input

hm	6. oct 2007		rev 1.2
	added pos and angle inputs and outputs
	night position and angle can now be configured
	any manual operation at night will cancel night operation

*)
END_FUNCTION_BLOCK

(* POU Building/Jalousie/blind_scene, ST *)
FUNCTION_BLOCK blind_scene
VAR_INPUT
	UP, DN : BOOL;
	S_IN : BYTE;
	pi, ai : BYTE;
	enable : BOOL;
	swrite : BOOL;
	scene : BYTE;
END_VAR
VAR_INPUT CONSTANT
END_VAR
VAR_OUTPUT
	QU, QD : BOOL;
	status : BYTE;
	po, ao : BYTE;
END_VAR
VAR RETAIN
	sx : ARRAY[0..15,0..2] OF BYTE;
END_VAR
VAR_TEMP
	x : BYTE;

END_VAR

(*
version 1.1	29. jan 2008
programmer 	hugo
tested by		tobias


*)
(* delete all bits except the lower 4 of scene *)
x := scene AND 16#0F;

IF enable AND sx[x,2] > 0 AND UP AND DN THEN
	po := sx[x,0];
	ao := sx[x,1];
	status := 160 + x;  (* Status number is 160 to 175 for the 16 scenes *)
	QU := TRUE;
	QD := TRUE;
ELSE
	QU := UP;
	QD := DN;
	status := S_IN;
	po := pi;
	ao := ai;
END_IF;

(* write scene if necessary *)
IF swrite THEN
	status := 176;		(* write scene *)
	sx[x,0] := pi;
	sx[x,1] := ai;
	IF enable THEN sx[x,2] := 1; ELSE sx[x,2] := 0; END_IF; (* if sx[x,2] = 0 the scene is disabled *)
END_IF;


(* revision history
hm	24. oct 2007	rev 1.0
	original release

hm		29.1.2008	rev 1.1
	replaced shr/shl with and for better performance
*)
END_FUNCTION_BLOCK

(* POU Building/Jalousie/blind_security, ST *)
FUNCTION_BLOCK blind_security
VAR_INPUT
	UP, DN : BOOL;
	S_IN : BYTE;
	pi, ai : BYTE;
	FIRE : BOOL;
	Wind : BOOL;
	Alarm : BOOL;
	Door : BOOL;
	Rain : BOOL;
END_VAR
VAR_INPUT CONSTANT
	Alarm_UP : BOOL := TRUE;
	WIND_UP :BOOL := TRUE;
	RAIN_UP : BOOL := FALSE;
END_VAR
VAR_OUTPUT
	QU, QD : BOOL;
	status : BYTE;
	po, ao : BYTE;
END_VAR
VAR
END_VAR

(*
version 1.2	12. feb 2008
programmer 	hugo
tested by		tobias


*)
IF Fire THEN
	QU := TRUE;
	QD := FALSE;
	status := 111;
ELSIF Wind THEN
	QU := Wind_up;
	QD := NOT wind_up;
	status := 112;
ELSIF alarm THEN
	QU := Alarm_up;
	QD := NOT Alarm_up;
	status := 113;
ELSIF Door THEN
	QU := TRUE;
	QD := FALSE;
	status := 114;
ELSIF Rain AND NOT (up XOR dn) THEN
	QU := rain_up;
	QD := NOT rain_up;
	status := 115;
ELSE
	QU := UP;
	QD := DN;
	status := S_IN;
	po := pi;
	ao := ai;
END_IF;


(* revision history
hm	29. sep 2007	rev 1.0
	original release

hm	6. oct 2007		rev 1.1
	added pos and angle inputs and outputs
	manual will override rain position
	alarm position can now be configured

hm		12. feb. 2008	rev 1.2
	added config variables rain_up and wind_up
	position for rain and wind is now configurable
*)
END_FUNCTION_BLOCK

(* POU Building/Jalousie/BLIND_SHADE, ST *)
FUNCTION_BLOCK BLIND_SHADE
VAR_INPUT
	UP, DN : BOOL;
	S_IN : BYTE;
	pi, ai : BYTE;
	enable : BOOL;
	sun : BOOL;
	dtin : DT;
	sunrise, sunset : TOD;
	sun_hor, sun_ver : REAL;
END_VAR
VAR_INPUT CONSTANT
	sunrise_offset : TIME := T#1h;
	sunset_preset : TIME := T#1h;
	direction : REAL := 180;
	angle_offset : REAL := 80;
	slat_width : REAL := 80;
	Slat_spacing : REAL := 60;
	Shade_delay : TIME := T#60s;
END_VAR
VAR_OUTPUT
	QU, QD : BOOL;
	status : BYTE;
	po, ao : BYTE;
END_VAR
VAR
	angle: REAL;
	sun_delay : TOF;
END_VAR

(*
version 1.2	24 nov 2007
programmer 	hugo
tested by		tobias


*)
(* the input sun is sent through tof which will delay the shade for the time shade_delay *)
sun_delay(IN := sun, PT := shade_delay);

IF UP AND DN AND enable AND sun_delay.Q AND sun_hor > direction - angle_offset AND sun_hor < direction + angle_offset AND
	DT_TO_TOD(dtin) > sunrise + sunrise_offset AND DT_TO_TOD(dtin) < sunset - sunset_preset THEN
	status := 151;
	QU := UP;
	QD := DN;
	(* position is fully down *)
	po := 0;
	(* shading is active now calculate the slat angle *)
	(* calculate the max angle for the blind *)
	angle := deg(ATAN(slat_spacing / slat_width));
	(* check if sun angle is between 0 and max angle *)
	IF sun_ver > 0 AND sun_ver < angle THEN
		angle := sun_ver + deg(ACOS(COS(Rad(sun_ver))*slat_spacing / Slat_width));
		ao := INT_TO_BYTE(LIMIT(0,TRUNC(angle * 255 / 90), 255));
	ELSE
		ao := 255;
	END_IF;
ELSE
	QU := UP;
	QD := DN;
	po := pi;
	ao := ai;
	status := S_IN;
END_IF;

(* revision history
hm	15 oct. 2007	rev 1.0
	original version

hm	19. oct 2007	rev 1.1
	manual mode was not detected because outputs were checked and not inputs UP and DN

hm	24. nov 2007	rev 1.2
	added shade_delay to avoid constant up and down if sun is out parcially
*)
END_FUNCTION_BLOCK

(* POU Mathematical/DEG, ST *)
FUNCTION DEG : REAL
VAR_INPUT
	rad : REAL;
END_VAR
VAR
END_VAR
VAR
END_VAR

(*
version 1.1	16 oct 2007
programmer 	hugo
tested by		tobias

this function converts degrees into Radiant
execution time on wago 750 - 841 =  10  us
*)
deg := modR(57.29577951308232 * Rad, 360);

(* revision history
hm	4. aug 2006		rev 1.0
	original version

hm 	16. oct 2007	rev 1.1
	added modr statement which prohibits deg to become bigger than 360

*)
END_FUNCTION

(* POU Mathematical/RAD, ST *)
FUNCTION RAD : REAL
VAR_INPUT
	deg : REAL;
END_VAR
VAR
END_VAR

(*
version 1.0	4 aug 2006
programmer 	hugo
tested by	tobias

this function converts Radiant to degrees

*)
Rad := modR(0.0174532925199433 * deg,PI2);

(* revision history
hm	4. aug 2006
	original version

hm 	16. oct 2007
	added modr statement which prohibits rad to become bigger than 2PI

*)
END_FUNCTION

(* POU Mathematical/MODR, ST *)
FUNCTION MODR : REAL
VAR_INPUT
	in : REAL;
	divi : REAL;
END_VAR

VAR
END_VAR

(*
version 1.1	4 aug 2006
programmer 	hugo
tested by		tobias

this is a modulo funtion for real numbers
modr(5.5,2.5) = 0.5

*)
IF divi = 0 THEN
	modR := 0;
ELSE
	modR := in - TRUNC(in / divi) * divi;
END_IF;

(* revision history

hm 4.8.2006	rev 1.0

hm 28.1.2007	rev 1.1
	modr(x,0) will deliver the result 0

*)
END_FUNCTION

(* POU Device Drivers/IRTRANS_1, ST *)
FUNCTION_BLOCK IRTRANS_1
VAR_INPUT CONSTANT
	device_code : STRING;
	key_code : STRING;
END_VAR
VAR_INPUT
	cmd : BOOL;
END_VAR
VAR_IN_OUT
	device : STRING;
	key : STRING;
END_VAR
VAR_OUTPUT
	Q : BOOL;
END_VAR
VAR
END_VAR

(*
	version 1.0	2 jan 2008
	programmer 	hugo
	tested BY		tobias

*)
IF cmd AND device_code = device AND key_code = key THEN
	Q := TRUE;
ELSE
	Q := FALSE;
END_IF;

(* revision history
hm	2. jan 2008		rev 1.0
	original version

*)
END_FUNCTION_BLOCK

(* POU Device Drivers/IRTRANS_4, ST *)
FUNCTION_BLOCK IRTRANS_4
VAR_INPUT CONSTANT
	device_code : STRING;
	key_code_0 : STRING;
	key_code_1 : STRING;
	key_code_2 : STRING;
	key_code_3 : STRING;
END_VAR
VAR_INPUT
	cmd : BOOL;
END_VAR
VAR_IN_OUT
	device : STRING;
	key : STRING;
END_VAR
VAR_OUTPUT
	Q0, Q1, Q2, Q3 : BOOL;
END_VAR
VAR
END_VAR

(*
	version 1.0	2 jan 2008
	programmer 	hugo
	tested BY		tobias

*)
Q0 := FALSE;
Q1 := FALSE;
Q2 := FALSE;
Q3 := FALSE;
IF cmd AND device_code = device THEN
	IF key = key_code_0 THEN q0 := TRUE;
	ELSIF key = key_code_1 THEN q1 := TRUE;
	ELSIF key = key_code_2 THEN q2 := TRUE;
	ELSIF key = key_code_3 THEN q3 := TRUE;
	END_IF;
END_IF;

(* revision history
hm	2. jan 2008		rev 1.0
	original version

*)
END_FUNCTION_BLOCK

(* POU Device Drivers/IRTRANS_8, ST *)
FUNCTION_BLOCK IRTRANS_8
VAR_INPUT CONSTANT
	device_code : STRING;
	key_code_0 : STRING;
	key_code_1 : STRING;
	key_code_2 : STRING;
	key_code_3 : STRING;
	key_code_4 : STRING;
	key_code_5 : STRING;
	key_code_6 : STRING;
	key_code_7 : STRING;
END_VAR
VAR_INPUT
	cmd : BOOL;
END_VAR
VAR_IN_OUT
	device : STRING;
	key : STRING;
END_VAR
VAR_OUTPUT
	Q0, Q1, Q2, Q3, Q4, Q5, Q6, Q7 : BOOL;
END_VAR
VAR
END_VAR

(*
	version 1.0	2 jan 2008
	programmer 	hugo
	tested BY		tobias

*)
Q0 := FALSE;
Q1 := FALSE;
Q2 := FALSE;
Q3 := FALSE;
Q4 := FALSE;
Q5 := FALSE;
Q6 := FALSE;
Q7 := FALSE;
IF cmd AND device_code = device THEN
	IF key = key_code_0 THEN q0 := TRUE;
	ELSIF key = key_code_1 THEN q1 := TRUE;
	ELSIF key = key_code_2 THEN q2 := TRUE;
	ELSIF key = key_code_3 THEN q3 := TRUE;
	ELSIF key = key_code_4 THEN q4 := TRUE;
	ELSIF key = key_code_5 THEN q5 := TRUE;
	ELSIF key = key_code_6 THEN q6 := TRUE;
	ELSIF key = key_code_7 THEN q7 := TRUE;
	END_IF;
END_IF;

(* revision history
hm	2. jan 2008		rev 1.0
	original version

*)
END_FUNCTION_BLOCK

(* POU Device Drivers/IRTRANS_DECODE, ST *)
FUNCTION_BLOCK IRTRANS_DECODE
VAR_INPUT
	buffer : POINTER TO ARRAY[0..32000] OF BYTE;
END_VAR
VAR_IN_OUT
	length : DINT;
END_VAR
VAR_OUTPUT
	cmd : BOOL;
	device : STRING;
	key : STRING;
	error : BOOL;
END_VAR
VAR
	pt : POINTER TO BYTE;
	i : INT;
	stop : INT;
END_VAR

(*
	version 1.0	2 jan 2008
	programmer 	hugo
	tested BY		tobias

*)
(* do nothing if the buffer is empty *)
IF length > 0 THEN
	i := 0;
	error := TRUE;
	stop := DINT_TO_INT(length) - 2;
	(* read characters before first comma and store in device *)
	pt := ADR(device);
	WHILE i < stop DO
		IF buffer^[i] = 44 THEN EXIT; END_IF;
		pt^ := buffer^[i];
		pt := pt + 1;
		i := i + 1;
	END_WHILE;
	(* terminate the device string *)
	pt^ := 0;
	(* read after first comma and store in key *)
	i := i + 1;
	pt := ADR(key);
	WHILE i < stop DO
		pt^ := buffer^[i];
		pt := pt + 1;
		i := i + 1;
	END_WHILE;
	(* terminate the key string *)
	pt^:= 0;
	(* check if last two characters are $R$N 13, 10 *)
	IF buffer^[i] <> 13 AND buffer^[i+1] <> 10 THEN	RETURN;	END_IF;
	(* check if device and key are present *)
	IF LEN(device) = 0 OR LEN(key) = 0 THEN RETURN; END_IF;
	(* a valid transmission has been received *)
	cmd := TRUE;
	error := FALSE;
	(* clear the input buffer to allow the next transmission to occur *)
	length := 0;
ELSE
	error := FALSE;
	cmd := FALSE;
END_IF;


(* revision history
hm	2. jan 2008		rev 1.0
	original version

*)
END_FUNCTION_BLOCK

(* POU Engineering/conversion/length, ST *)
FUNCTION_BLOCK length
VAR_INPUT
	m : REAL;
	p : REAL;
	in : REAL;
	ft : REAL;
	yd : REAL;
	mile : REAL;
	sm : REAL;
	fm : REAL;
END_VAR
VAR_OUTPUT
	Ym : REAL;
	Yp : REAL;
	Yin : REAL;
	Yft : REAL;
	Yyd : REAL;
	Ymile : REAL;
	Ysm : REAL;
	Yfm : REAL;
END_VAR
VAR
END_VAR

(*
version 1.0	27 mar 2007
programmer 	hugo
tested by		oscat

this function converts different length units
any unused input can simply be left open.
different inputs connected at the same time will be added up.

*)
Ym :=	m
		+ p * 0.000376065
		+ in * 0.0254
		+ ft * 0.3048
		+ yd * 0.9144
		+ mile * 1609.344
		+ sm * 1852
		+ fm * 1.829;
Yp := Ym / 0.000376065;
Yin := Ym / 0.0254;
Yft := Ym / 0.3048;
Yyd := Ym / 0.9144;
Ymile := Ym / 1609.344;
Ysm := Ym / 1852;
Yfm := Ym / 1.829;

(*
Länge Meter m SI-Basiseinheit
Astronomische Einheit* AE 1 AE = 149,597 870 · E9 m
Parsec pc 1 pc = 206265 AE = 30,857 · E15 m
Lichtjahr Lj 1 Lj = 9,460 530 · E15 m = 63240 AE = 0,306 59 pc
Ångström Å 1 Å = E–l0 m
typograph. Punkt p 1 p = 0,376 065 mm • im Druckereigewerbe
inch** in 1 in = 2,54 · E–2 m = 25,4 mm***
foot ft 1 ft = 0,3048 m = 30,48 cm
yard yd 1 yd = 0,9144 m
mile mile 1 mile = 1609,344 m
Internat. Seemeile sm 1 sm = 1852 m
Fathom fm 1 fm = 1,829 m • in der Seeschifffahrt

*)
END_FUNCTION_BLOCK

(* POU Engineering/automation/DRIVER_1, ST *)
FUNCTION_BLOCK DRIVER_1
VAR_INPUT CONSTANT
	Toggle_Mode : BOOL;
	Timeout : TIME;
END_VAR
VAR_INPUT
	SET : BOOL;
	IN : BOOL;
	RST : BOOL;
END_VAR
VAR_OUTPUT
	Q : BOOL;
END_VAR
VAR
	off : TON;
	edge: BOOL;
END_VAR

(*
version 1.0	2 jan 2008
programmer 	hugo
tested by		tobias

driver_1 is a multi purpose driver.
a rising edge on in sets the output high if toggle is flase. while toggle is true, a rising edge on in toggles the output Q.
if a timeout is specified the output q will be reset to false automatically after the timeout has elapsed.
a asynchronous reset and set will force the output high or low respectively.

*)
IF off.Q THEN Q := FALSE; END_IF;
IF rst THEN
	Q := FALSE;
ELSIF set THEN
	Q := TRUE;
ELSIF IN AND NOT edge THEN
	IF toggle_mode THEN q := NOT Q; ELSE q := TRUE; END_IF;
END_IF;
edge := in;
IF timeout > t#0s THEN off(in := Q, PT := Timeout); END_IF;


(* revision history
hm	2. jan 2008		rev 1.0
	original version

*)
END_FUNCTION_BLOCK

(* POU Engineering/automation/DRIVER_4, ST *)
FUNCTION_BLOCK DRIVER_4
VAR_INPUT CONSTANT
	Toggle_Mode : BOOL;
	Timeout : TIME;
END_VAR
VAR_INPUT
	SET : BOOL;
	IN0, IN1, IN2, IN3 : BOOL;
	RST : BOOL;
END_VAR
VAR_OUTPUT
	Q0, Q1, Q2, Q3 : BOOL;
END_VAR
VAR
	d0, d1, d2, d3 : DRIVER_1;
END_VAR

(*
version 1.0	2 jan 2008
programmer 	hugo
tested by		tobias

driver_4 is a 4 channel multi purpose driver.
a rising edge on in? sets the output Q? high if toggle_mode is flase. while toggle_mode is true, a rising edge on in? toggles the output Q?.
if a timeout is specified the output Q? will be reset to false automatically after the timeout has elapsed.
a asynchronous reset and set will force the output high or low respectively.
an asynchronous set will force all outputs high simultaneously

*)
D0(Set:=set, in:=in0, rst:=rst, toggle_mode:=toggle_mode, timeout:=timeout);
D1(Set:=set, in:=in1, rst:=rst, toggle_mode:=toggle_mode, timeout:=timeout);
D2(Set:=set, in:=in2, rst:=rst, toggle_mode:=toggle_mode, timeout:=timeout);
D3(Set:=set, in:=in3, rst:=rst, toggle_mode:=toggle_mode, timeout:=timeout);
Q0 := D0.Q;
Q1 := D1.Q;
Q2 := D2.Q;
Q3 := D3.Q;


(* revision history
hm	2. jan 2008		rev 1.0
	original version

*)
END_FUNCTION_BLOCK

(* POU Engineering/automation/FT_Profile, ST *)
FUNCTION_BLOCK FT_Profile
VAR_INPUT
	K : REAL := 1;
	O : REAL := 0;
	M : REAL := 1;
	E : BOOL;
END_VAR
VAR_INPUT CONSTANT
	value_0 : REAL;
	time_1 : TIME;
	value_1 : REAL;
	time_2 : TIME;
	value_2 : REAL;
	time_3 : TIME;
	value_3 : REAL;
	time_10 : TIME;
	value_10 : REAL;
	time_11 : TIME;
	value_11 : REAL;
	time_12 : TIME;
	value_12 : REAL;
	time_13 : TIME;
	value_13 : REAL;
END_VAR
VAR_OUTPUT
	Y : REAL;
	RUN : BOOL;
	ET : TIME;
END_VAR
VAR
	tx : TIME;
	edge : BOOL;
	state: BYTE;
	ta: TIME;
	tb: TIME;
	t0 : TIME;
	temp: REAL;
	va: REAL;
	vb: REAL;
END_VAR

(*
version 1.1	15 sep 2007
programmer 	tobias
tested by		hugo

FT_Profile generates an output signal which is defined by values over a time scale.
the different values are connected by ramps between the individual values.
a rising edge on E starts the output signal generation and E = True can delay time_3 / value_3 as long as it stays true.
an additional multiplier K can be used to multiply the output and an offset O can be added to the output dynamically.
*)
(* read system time *)
tx := DWORD_TO_TIME(T_PLC_MS());

(* determine start condition *)
IF E AND NOT edge THEN
	RUN := TRUE;
	ET := t#0s;
	t0 := tx;
	ta := tx;
	tb := multime(time_1, M);
	va := value_0;
	vb := value_1;
	temp := value_0;
	state := 1;
END_IF;
edge := E;

(* generate startup profile *)
IF run THEN
	CASE state OF
		1:	IF tx - ta >= tb THEN
				ta := ta + tb;
				tb := multime(time_2 - time_1, M);
				va := value_1;
				vb := value_2;
				temp := value_1;
				state := 2;
			ELSE
				temp := ((vb - va) * TIME_TO_REAL(tx - ta) / TIME_TO_REAL(tb) + va);
			END_IF;
		2:	IF tx - ta >= tb THEN
				ta := ta + tb;
				tb := multime(time_3 - time_2, M);
				va := value_2;
				vb := value_3;
				temp := value_2;
				state := 3;
			ELSE
				temp := ((vb - va) * TIME_TO_REAL(tx - ta) / TIME_TO_REAL(tb) + va);
			END_IF;
		3:	IF tx - ta >= tb THEN
				ta := ta + tb;
				tb := multime(time_10 - time_3, M);
				va := value_3;
				vb := value_10;
				temp := value_3;
				state := 4;
			ELSE
				temp := ((vb - va) * TIME_TO_REAL(tx - ta) / TIME_TO_REAL(tb) + va);
			END_IF;
		4 :	IF tx - ta >= tb THEN
				ta := ta + tb;
				tb := multime(time_11 - time_10, M);
				va := value_10;
				vb := value_11;
				temp := value_10;
				IF E THEN state := 5; ELSE state := 6; END_IF;
			ELSE
				temp := ((vb - va) * TIME_TO_REAL(tx - ta) / TIME_TO_REAL(tb) + va);
			END_IF;
		5:	(* extend the signal while E is true *)
			IF E THEN
				ta := tx;
			ELSE
				state := 6;
			END_IF;
		6:	IF tx - ta >= tb THEN
				ta := ta + tb;
				tb := multime(time_12 - time_11, M);
				va := value_11;
				vb := value_12;
				temp := value_11;
				state := 7;
			ELSE
				temp := ((vb - va) * TIME_TO_REAL(tx - ta) / TIME_TO_REAL(tb) + va);
			END_IF;
		7:	IF tx - ta >= tb THEN
				ta := ta + tb;
				tb := multime(time_13 - time_12, M);
				va := value_12;
				vb := value_13;
				temp := value_12;
				state := 8;
			ELSE
				temp := ((vb - va) * TIME_TO_REAL(tx - ta) / TIME_TO_REAL(tb) + va);
			END_IF;
		8:	IF tx - ta >= tb THEN
				temp := value_13;
				run := FALSE;
			ELSE
				temp := ((vb - va) * TIME_TO_REAL(tx - ta) / TIME_TO_REAL(tb) + va);
			END_IF;
	END_CASE;
	Y := temp * K + O;
	ET := tx - t0;
END_IF;

(* revision history
hm	27 feb 2007		rev 1.0
	original version

hm	15. sep2007		rev 1.1
	replaced Time() with T_PLC_MS for compatibility and performance reasons

*)
END_FUNCTION_BLOCK

(* POU Engineering/automation/inc_dec, ST *)
FUNCTION_BLOCK inc_dec
VAR_INPUT
	CHa : BOOL;
	CHb : BOOL;
	RST : BOOL := 0;
END_VAR
VAR_OUTPUT
	dir : BOOL;
	cnt : INT;
END_VAR
VAR
	edgea : BOOL := 0;
	clk: BOOL;
	clka: BOOL;
	clkb: BOOL;
	edgeb: BOOL;
	axb: BOOL;
END_VAR

(*
	version 1.0	4 aug 2006
	programmer 	oscat
	tested BY		oscat

incremental decoder with quadruple accuracy.
2 pulses for each channel are created for each directional pulse.
*)
axb := cha XOR chb;

(* create pulses for channel a *)
clka := cha XOR edgea;
edgea := cha;

clkb := chb XOR edgeb;
edgeb := chb;

(* create pulses for both channels *)
clk := clka OR clkb;

(* set the direction output *)
IF axb AND clka THEN dir := TRUE; END_IF;
IF axb AND clkb THEN dir := FALSE; END_IF;

(* increment or decrement the counter *)
IF clk AND dir THEN cnt := cnt + 1; END_IF;
IF clk AND NOT dir THEN cnt := cnt -1; END_IF;

(* reset the counter if rst active *)
IF rst THEN cnt := 0; END_IF;
END_FUNCTION_BLOCK

(* POU Engineering/automation/parset, ST *)
FUNCTION_BLOCK parset
VAR_INPUT
	A0, A1 : BOOL;
END_VAR
VAR_INPUT CONSTANT
	X01, X02, X03, X04 : REAL;
	X11, X12, X13, X14 : REAL;
	X21, X22, X23, X24 : REAL;
	X31, X32, X33, X34 : REAL;
	TC : TIME;
END_VAR
VAR_OUTPUT
	P1, P2, P3, P4 : REAL;
END_VAR
VAR
	X : ARRAY[0..3,1..4] OF REAL;
	S1, S2, S3, S4 : REAL;
	tx, last : DWORD;
	start : BOOL;
	set : BYTE;
	init: BOOL;
END_VAR

(*
version 1.0	2 nov 2007
programmer 	hugo
tested by		tobias

parset selects on of 4 parameter sets adressed by the inputs A0 and A1. if TC is specified, the change of the outputs
is ramped by the time tc
*)
(* read system_time *)
tx := T_PLC_MS();

(* init sequence *)
IF NOT init THEN
	set.0 := NOT A0;
	init := TRUE;
	X[0,1] := X01;
	X[0,2] := X02;
	X[0,3] := X03;
	X[0,4] := X04;
	X[1,1] := X11;
	X[1,2] := X12;
	X[1,3] := X13;
	X[1,4] := X14;
	X[2,1] := X21;
	X[2,2] := X22;
	X[2,3] := X23;
	X[2,4] := X24;
	X[3,1] := X31;
	X[3,2] := X32;
	X[3,3] := X33;
	X[3,4] := X34;
	P1 := X01;
	P2 := X02;
	P3 := X03;
	P4 := X04;
END_IF;

(* check for input change *)
IF (A0 XOR set.0) OR (A1 XOR set.1) THEN
	(* a new set is selected *)
	set.0 := A0;
	set.1 := A1;
	IF tc > t#0s THEN
		start := TRUE;
		last := tx;
		(* save the step speed for the output changes in S *)
		S1 := (X[set,1] - P1)/TIME_TO_DWORD(tc);
		S2 := (X[set,2] - P2)/TIME_TO_DWORD(tc);
		S3 := (X[set,3] - P3)/TIME_TO_DWORD(tc);
		S4 := (X[set,4] - P4)/TIME_TO_DWORD(tc);
	END_IF;
ELSIF start AND tx - last < TIME_TO_DWORD(tc) THEN
	(* ramp the outputs to the new value *)
	P1 := X[set,1] - S1*(TIME_TO_DWORD(Tc) - tx + last);
	P2 := X[set,2] - S2*(TIME_TO_DWORD(Tc) - tx + last);
	P3 := X[set,3] - S3*(TIME_TO_DWORD(Tc) - tx + last);
	P4 := X[set,4] - S4*(TIME_TO_DWORD(Tc) - tx + last);
ELSE
	(* make sure outputs match the correct set values *)
	start := FALSE;
	P1 := X[set,1];
	P2 := X[set,2];
	P3 := X[set,3];
	P4 := X[set,4];
END_IF;

(* revision history
hm		2.11.2007		rev 1.0
	original version

*)
END_FUNCTION_BLOCK

(* POU Engineering/automation/parset2, ST *)
FUNCTION_BLOCK parset2
VAR_INPUT
	X : REAL;
END_VAR
VAR_INPUT CONSTANT
	X01, X02, X03, X04 : REAL;
	X11, X12, X13, X14 : REAL;
	X21, X22, X23, X24 : REAL;
	X31, X32, X33, X34 : REAL;
	L1, L2, L3 : REAL;
	TC : TIME;
END_VAR
VAR_OUTPUT
	P1,P2,P3,P4 : REAL;
END_VAR
VAR
	Pset : parset;
	init: BOOL;
END_VAR

(*
version 1.0	3 nov 2007
programmer 	hugo
tested by	tobias

parset2 selects on of 4 parameter sets depending on the value of X. if TC is specified, the change of the outputs
is ramped by the time TC
*)
(* init sequence *)
IF NOT init THEN
	init := TRUE;
	pset(TC:=TC, X01:=X01, X02:=X02, X03:=X03, X04:=X04, X11:=X11, X12:=X12, X13:=X13, X14:=X14, X21:=X21, X22:=X22, X23:=X23, X24:=X24, X31:=X31, X32:=X32, X33:=X33, X34:=X34);
END_IF;
IF ABS(X) < L1 THEN
	pset(A0 := FALSE, A1 := FALSE);
ELSIF ABS(X) < L2 THEN
	pset(A0 := TRUE, A1 := FALSE);
ELSIF ABS(x) < L3 THEN
	pset(A0 := FALSE, A1 := TRUE);
ELSE
	pset(A0 := TRUE, A1 := TRUE);
END_IF;
P1 := pset.P1;
P2 := pset.P2;
P3 := pset.P3;
P4 := pset.P4;

(* revision history
hm		3.11.2007		rev 1.0
	original version

*)
END_FUNCTION_BLOCK

(* POU Engineering/automation/SIGNAL, ST *)
FUNCTION_BLOCK SIGNAL
VAR_INPUT
	IN : BOOL;
	SIG : BYTE;
	TS : TIME;
END_VAR
VAR_OUTPUT
	Q : BOOL;
END_VAR
VAR
	tx: DWORD;
	step: BYTE;
END_VAR
VAR CONSTANT
	one : BYTE := 1;
END_VAR

(*
version 1.0	13 dec 2007
programmer 	hugo
tested by		tobias

this function generates an output signal according to a bit pattern SIG.
the patter is shifted to the output in time steps of TS.
ts defaults to 128 ms if not specified.
*)
IF in THEN
	(* an alarm is present read system time first *)
	tx := T_PLC_MS();
	(* calculate the step counter which is the lowest 3 bits of (time / ts) *)
	IF ts > t#0s THEN
		step := DWORD_TO_BYTE(tx / TIME_TO_DWORD(ts) AND 16#0000_0007);
	ELSE
		step := DWORD_TO_BYTE(SHR(tx,7) AND 16#0000_0007);
	END_IF;
	(* convert the value 0-7 in step into one bit only (bit 0-7) *)
	step := SHL(one,step);
	(* generate the output signal *)
	Q := (step AND sig) > 0;
ELSE
	Q := FALSE;
END_IF;

(* revision history
hm	13.12.2007		rev 1.0
	original version

*)
END_FUNCTION_BLOCK

(* POU Engineering/automation/SIGNAL_4, ST *)
FUNCTION_BLOCK SIGNAL_4
VAR_INPUT
	IN1 : BOOL;
	IN2 : BOOL;
	IN3 : BOOL;
	IN4 : BOOL;
	TS : TIME;
END_VAR
VAR_INPUT CONSTANT
	S1 : BYTE := 2#1111_1111;
	S2 : BYTE := 2#1111_0000;
	S3 : BYTE := 2#1010_1010;
	S4 : BYTE := 2#1010_0000;
END_VAR
VAR_OUTPUT
	Q : BOOL;
END_VAR
VAR
	sig : SIGNAL;
END_VAR

(*
version 1.0	13 dec 2007
programmer 	hugo
tested by		tobias

this function generates one out of 4 signals specified by bit patterns S1 .. S4.
the selected pattern will be shifted with the step time TS.
In1 has higher priority then In2 which has higher priority then IN3 and in4 has the lowest priority.
ts defaults to 128 ms if not specified.
*)
(* an alarm is present read system time first *)
(* check if an alarm is present if yes set sig to the alarm pattern otherwise exit the routine *)
IF in1 THEN
	sig(in := TRUE, sig := s1, TS := TS);
ELSIF in2 THEN
	sig(in := TRUE, sig := s2, TS := TS);
ELSIF in3 THEN
	sig(in := TRUE, sig := s3, TS := TS);
ELSIF in4 THEN
	sig(in := TRUE, sig := s4, TS := TS);
ELSE
	sig(in := FALSE);
END_IF;

(* set the output *)
Q := sig.Q;


(* revision history
hm	13.12.2007		rev 1.0
	original version

*)
END_FUNCTION_BLOCK

(* POU Engineering/automation/tune, ST *)
FUNCTION_BLOCK tune
VAR_INPUT
	SET : BOOL;
	SU, SD : BOOL;
	RST : BOOL;
END_VAR
VAR_INPUT CONSTANT
	SS : REAL := 0.1;
	Limit_L : REAL := 0;
	LIMIT_H : REAL := 100;
	RST_val : REAL := 0;
	SET_val : REAL := 100;
	T1 : TIME := T#500ms;
	T2 : TIME := T#2s;
	S1 : REAL := 2;
	S2 : REAL := 10;
END_VAR
VAR_OUTPUT
	Y : REAL;
END_VAR
VAR
	tx : DWORD;
	start, start2 : DWORD;
	state : INT;
	in : BOOL;
	step : REAL;
	speed : REAL;
	Y_start : REAL;
	Y_start2: REAL;
END_VAR

(*
version 1.0	3 nov 2007
programmer 	hugo
tested by	tobias

tune generates an output signal which is set by input switches.
up to 4 switsches can be used to tune the signal up or down.

*)
(* read system time *)
tx := T_PLC_MS();

IF rst THEN
	Y := RST_val;
	state := 0;
ELSIF set THEN
	Y := SET_val;
	state := 0;
ELSIF state > 0 THEN
	(* key has been pushed state machine operating *)
	(* first read the correct input *)
	IF state = 1 THEN
		(* step up *)
		in := su;
	ELSE
		(* step down *)
		in := sd;
	END_IF;
	(* check for single step operation *)
	IF NOT in AND tx - start <= TIME_TO_DWORD(T1) THEN
		Y := Y_start + step;
		state := 0;
	(* check if fast ramp needs to be generated *)
	ELSIF in AND tx - start >= TIME_TO_DWORD(T2) THEN
		Y := Y_start2 + (tx - start2) * s2 / speed;
	(* check if slow ramp needs to be generated *)
	ELSIF in AND tx - start >= TIME_TO_DWORD(T1) THEN
		Y := Y_start + (tx - start - TIME_TO_DWORD(T1)) * S1 / speed;
		start2 := tx;
		Y_start2 := Y;
	ELSIF NOT in THEN
		state := 0;
	END_IF;
ELSIF su THEN
	(* slow step up *)
	state := 1;
	start := tx;
	step := ss;
	speed := 1000;
	Y_start := Y;
ELSIF sd THEN
	(* slow step down *)
	state := 2;
	start := tx;
	step := -ss;
	speed := -1000;
	Y_start := Y;
END_IF

(* make sure output does not exceed limits *)
Y := LIMIT(LIMIT_L, Y, LIMIT_H);

(* revision history
hm		3.11.2007		rev 1.0
	original version

*)
END_FUNCTION_BLOCK

(* POU Engineering/conversion/speed, ST *)
FUNCTION_BLOCK speed
VAR_INPUT
	ms : REAL;
	kmh : REAL;
	kn : REAL;
	mh : REAL;
END_VAR
VAR_OUTPUT
	Yms : REAL;
	Ykmh : REAL;
	Ykn : REAL;
	Ymh : REAL;
END_VAR
VAR
END_VAR

(*
version 1.0	27 mar 2007
programmer 	hugo
tested by		oscat

this function converts different speed units
any unused input can simply be left open.
different inputs connected at the same time will be added up.

*)
Yms := ms +
		kmh /3.6 +
		kn * 0.5144444 +
		mh * 0.44704;
Ykmh := Yms *3.6;
Ykn := Yms / 0.5144444;
Ymh := Yms / 0.44704;

(*
Geschwindigkeit Meter durch Sekunde m/s 1 m/s = 3,6 km/h
km durch (pro) Stunde, nicht „Stundenkilometer“ verwenden
Knoten kn 1 kn = 1 sm/h = 0,5144 m/s

*)
END_FUNCTION_BLOCK

(* POU Engineering/automation/tune2, ST *)
FUNCTION_BLOCK tune2
VAR_INPUT
	SET : BOOL;
	SU, SD : BOOL;
	FU, FD : BOOL;
	RST : BOOL;
END_VAR
VAR_INPUT CONSTANT
	SS : REAL := 0.1;
	FS : REAL := 5;
	Limit_L : REAL := 0;
	LIMIT_H : REAL := 100;
	RST_val : REAL := 0;
	SET_val : REAL := 100;
	TR : TIME := T#500ms;
	S1 : REAL := 2;
	S2 : REAL := 10;
END_VAR
VAR_OUTPUT
	Y : REAL;
END_VAR
VAR
	tx : DWORD;
	start : DWORD;
	state : INT;
	in : BOOL;
	step : REAL;
	speed : REAL;
	Y_start : REAL;
END_VAR

(*
version 1.0	3 nov 2007
programmer 	hugo
tested by	tobias

tune2 generates an output signal which is set by input switches.
up to 4 switsches can be used to tune the signal up or down.

*)
(* read system time *)
tx := T_PLC_MS();

IF rst THEN
	Y := RST_val;
	state := 0;
ELSIF set THEN
	Y := SET_val;
	state := 0;
ELSIF state > 0 THEN
	(* key has been pushed state machine operating *)
	(* first read the correct input *)
	CASE state OF
		1 :	(* slow up *)
			in := su;
		2 :	(* slow down *)
			in := sd;
		3 :	(* fast up *)
			in := fu;
		4 :	(* fast down *)
			in := fd;
	END_CASE;
	(* check for single step operation *)
	IF NOT in AND tx - start <= TIME_TO_DWORD(TR) THEN
		Y := Y_start + step;
		state := 0;
	(* check if ramp needs to be generated *)
	ELSIF in AND tx - start >= TIME_TO_DWORD(TR) THEN
		Y := Y_start + (tx - start - TIME_TO_DWORD(TR)) * speed;
	ELSIF NOT in THEN
		state := 0;
	END_IF;
ELSIF su THEN
	(* slow step up *)
	state := 1;
	start := tx;
	step := ss;
	speed := s1 / 1000;
	Y_start := Y;
ELSIF sd THEN
	(* slow step down *)
	state := 2;
	start := tx;
	step := -ss;
	speed := -s1 / 1000;
	Y_start := Y;
ELSIF fu THEN
	(* fast step up *)
	state := 3;
	start := tx;
	step := fs;
	speed := s2 / 1000;
	y_start := Y;
ELSIF fd THEN
	(* fast step down *)
	state := 4;
	start := tx;
	step := -fs;
	speed := -s2 / 1000;
	y_start := Y;
END_IF

(* make sure output does not exceed limits *)
Y := LIMIT(LIMIT_L, Y, LIMIT_H);

(* revision history
hm		3.11.2007		rev 1.0
	original version

*)
END_FUNCTION_BLOCK

(* POU Engineering/control/control_set1, ST *)
FUNCTION_BLOCK control_set1
VAR_INPUT
	Kt : REAL;
	Tt : REAL;
	PI : BOOL;
	PID : BOOL;
END_VAR
VAR_INPUT CONSTANT
	P_K : REAL := 0.5;
	PI_K : REAL := 0.45;
	PI_TN : REAL := 0.83;
	PID_K : REAL := 0.6;
	PID_TN : REAL := 0.5;
	PID_TV : REAL := 0.125;
END_VAR
VAR_OUTPUT
	KP : REAL;
	TN : REAL;
	TV : REAL;
	KI : REAL;
	KD : REAL;
END_VAR
VAR
END_VAR

(*
version 1.0	4 nov 2007
programmer 	hugo
tested by	tobias

takahashi calculates controller parameters for P, PI and PID controllers based on the ziegler nichols method.

*)
IF pi AND PID THEN
	KP := 0;
	TN := 0;
	TV := 0;
ELSIF PID THEN
	KP := PID_K * Kt;
	TN := PID_TN * Tt;
	TV := PID_TV * Tt;
ELSIF PI THEN
	KP := PI_K * Kt;
	TN := PI_TN * Tt;
ELSE
	KP := P_K * Kt;
END_IF;

(* KI and KD are calculated *)
IF tn > 0 THEN KI := KP / TN; ELSE KI := 0; END_IF;
KD := KP * TV;

(* revision history
hm	4. nov 2007		rev 1.0
	original version

*)
END_FUNCTION_BLOCK

(* POU Engineering/control/control_set2, ST *)
FUNCTION_BLOCK control_set2
VAR_INPUT
	KS : REAL;
	TU : REAL;
	TG : REAL;
	PI : BOOL;
	PID : BOOL;
END_VAR
VAR_INPUT CONSTANT
	P_K : REAL := 1.0;
	PI_K : REAL := 0.9;
	PI_TN : REAL := 3.33;
	PID_K : REAL := 1.2;
	PID_TN : REAL := 2;
	PID_TV : REAL := 0.5;
END_VAR
VAR_OUTPUT
	KP : REAL;
	TN : REAL;
	TV : REAL;
	KI : REAL;
	KD : REAL;
END_VAR
VAR
	TX : REAL;
END_VAR

(*
version 1.0	4 nov 2007
programmer 	hugo
tested by	tobias

takahashi calculates controller parameters for P, PI and PID controllers based on the ziegler nichols method.

*)
IF TU > 0 AND KS > 0 THEN TX := TG/TU/KS; END_IF;
IF pi AND PID THEN
	KP := 0;
	TN := 0;
	TV := 0;
ELSIF PID THEN
	KP := PID_K * TX;
	TN := PID_TN * TU;
	TV := PID_TV * TU;
ELSIF PI THEN
	KP := PI_K * TX;
	TN := PI_TN * TU;
ELSE
	KP := P_K * TX;
END_IF;

(* KI and KD are calculated *)
IF TN > 0 THEN KI := KP / TN; ELSE KI := 0; END_IF;
KD := KP * TV;

(* revision history
hm	4. nov 2007		rev 1.0
	original version

*)
END_FUNCTION_BLOCK

(* POU Engineering/control/DEAD_BAND, ST *)
FUNCTION DEAD_BAND : REAL
VAR_INPUT
	X : REAL;
	L : REAL;
END_VAR
VAR
END_VAR

(*
version 1.0	2 nov 2007
programmer 	hugo
tested by		tobias

DEAD_BAND ist eine lineare Übertragungsfunktion mit Totzone. Die Funktion verschiebt den positiven Teil der Kurve um +L und den negativen Teil der Kurve um -L.
DEAD_BAND = X wenn Abs(X) > L wenn Abs(X) > L
DEAD_BAND = 0 wenn Abs(X) <= L

*)
IF ABS(x) > L THEN
	dead_band := X - sgn(x) * L;
ELSE
	dead_band := 0;
END_IF;

(* revision history
hm		2.11.07	rev 1.0
	original version
*)
END_FUNCTION

(* POU Mathematical/SGN, ST *)
FUNCTION SGN : INT
VAR_INPUT
	X : REAL;
END_VAR
VAR
END_VAR

(*
version 1.1	11 nov 2007
programmer 	hugo
tested by	tobias

sgn returns 0 when X = 0 , -1 when X < 1 and +1 when X > 1

*)
IF X > 0 THEN
	sgn := 1;
ELSIF X < 0 THEN
	sgn := -1;
ELSE
	sgn := 0;
END_IF;

(* revision histroy
hm	16. oct 2007	rev 1.0
	original version

hm	11. nov 2007	rev 1.1
	changed type of function from real to int
*)
END_FUNCTION

(* POU Engineering/control/dead_zone, ST *)
FUNCTION dead_zone : REAL
VAR_INPUT
	X : REAL;
	L : REAL;
END_VAR
VAR
END_VAR

(*
version 1.0	12 Feb 2007
programmer 	hugo
tested by		tobias

dead_zone2 is a linear transfer function which follows a linear function except for x is close to 0.
Y = X if abs(x) > L otherwise its 0.

*)
IF ABS(x) > L THEN
	dead_zone := X;
ELSE
	dead_zone := 0;
END_IF;
END_FUNCTION

(* POU Engineering/control/dead_zone2, ST *)
FUNCTION_BLOCK dead_zone2
VAR_INPUT
	X : REAL;
	L : REAL;
END_VAR
VAR_OUTPUT
	Y: REAL;
END_VAR
VAR
END_VAR

(*
version 1.0	12 Feb 2007
programmer 	hugo
tested by		tobias

dead_zone2 is a linear transfer function which follows a linear function except for x is close to 0.
Y = X if abs(x) > L.
for values of 0 +/. L a hysteresis function will hold the output at + or - L.

*)
IF ABS(x) > L THEN
	Y := X;
ELSIF Y > 0 THEN
	Y := L;
ELSE
	Y := -L;
END_IF;
END_FUNCTION_BLOCK

(* POU Engineering/control/FT_deriv, ST *)
FUNCTION_BLOCK FT_deriv
VAR_INPUT
	in : REAL;
	K : REAL := 1;
	run : BOOL := 1;
END_VAR
VAR_OUTPUT
	out : REAL;
END_VAR
VAR
	old: REAL;
	tx: DWORD;
	last: DWORD;
	init: BOOL;
END_VAR


(*
version 1.3	29 oct 2007
programmer 	hugo
tested by		tobias

FT_deriv calculates the derivate over the signal "in" with Faktor "K".
a run input enables or stops the calculation, if left unconnected its true and therfore the calculation is executed.
if K is not specified the default is 1.

*)
(* read system time *)
tx := T_PLC_US();

(* init on firsat startup *)
IF NOT init THEN
	init := TRUE;
	old := in;
	last := tx;
END_IF;
IF run AND tx - last > 0 THEN
	out := (in - old) / DWORD_TO_REAL(tx - last) * 1000000.0 * K;
	last := tx;
ELSE
	out := 0;
	last := tx;
END_IF;
old := in;


(*
hm 3.1.2007			rev 1.1
	added init code for startup
	set the default for K to 1

hm	15. sep 2007	rev 1.2
	replaced Time() with T_PLC_US for compatibility and performance reasons
	increased accuracy and work in microseconds internally

hm 29 oct 2007	rev 1.3
	prohibit calculation when tx - last = 0 to avoid division by 0 and increase accuracy on fast systems
*)
END_FUNCTION_BLOCK

(* POU Engineering/control/FT_IMP, ST *)
FUNCTION_BLOCK FT_IMP
VAR_INPUT
	in : REAL;
	T : TIME;
	K : REAL := 1;
END_VAR
VAR_OUTPUT
	out : REAL;
END_VAR
VAR
	t1 : FT_PT1;
END_VAR

(*
version 1.1	3 Jan 2007
programmer 	hugo
tested by		tobias

FT_IMP is 	an impulse filter (high pass filter) with the time T and factor K.
 
*)
T1(in:= in, T:=T);
out := (in - t1.out) * K;

(*
hm 3.1.2007	rev 1.1
	added factor K

*)
END_FUNCTION_BLOCK

(* POU Engineering/control/FT_PT1, ST *)
FUNCTION_BLOCK FT_PT1
VAR_INPUT
	in : REAL;
	T : TIME;
	K : REAL := 1;
END_VAR
VAR_OUTPUT
	out : REAL;
END_VAR
VAR
	last : DWORD;
	tx: DWORD;
	init: BOOL;
END_VAR

(*
version 1.7	5 jan 2008
programmer 	hugo
tested by		tobias

FT_PT1 is an low pass filter with a programmable time T and faktor K.
 
*)
(* read system time *)
tx := T_PLC_US();

(* startup initialisation *)
IF NOT init THEN
	last := tx;
	init := TRUE;
	out := K * in;
ELSIF T = t#0s THEN
	out := K * in;
ELSE
	out := out + (in * K - out) * (Tx - last) / TIME_TO_REAL(T) * 1E-3;
END_IF;
last := tx;

(*
hm 1.1.2007	rev 1.1
	corrected error while startup value was not correct
	for very small time values real output would run out of range.

hm 3.1.2007	rev 1.2
	corrected an error for falling edge failures.
	added output faktor K.

hm 27. 2. 2007	rev 1.3
	output will be input during init for definitive startup condition.

hm	15.9.2007	rev 1.4
	changed time() to T_PLC_US() for compatibilitxy resons
	increased internal accuracy to Microseconds instead of Milliseconds

hm	23. oct 2007	rev 1.5
	added out := in to the init statements

hm	30. nov 2007	rev 1.6
	changed out to be K * in during initialization

hm	5. jan 2008		rev 1.7
	improved code for better performance
*)
END_FUNCTION_BLOCK

(* POU Engineering/control/FT_PI, ST *)
FUNCTION_BLOCK FT_PI
VAR_INPUT
	actual, set_point, noise, offset, manual_in : REAL;
	Manual : BOOL;
	rst : BOOL := FALSE;
	int_band : REAL := 100;
	KP : REAL := 1.0;
	KI : REAL := 1.0;
	limit_L : REAL := -1000;
	limit_H : REAL := 1000;
END_VAR
VAR_INPUT CONSTANT
	int_limit_L : REAL := -1000;
	int_limit_H : REAL := 1000;
END_VAR
VAR_OUTPUT
	Y : REAL;
	DIFF : REAL;
	LIM, overflow : BOOL;
END_VAR
VAR
	integ : FT_INT;
END_VAR

(*
version 1.2	5 jan 2008
programmer 	hugo
tested by		tobias

FT_PI is a PI controller with manual functionality.
The PID controller works according to the fomula Y = e *(KP+ KI * INTEG(e) ) + offset, while e = set_point - actual.
a rst will reset all internal data, while a switch to manual will cause the controller to follow the function Y = manual_in + offset.
limit_h and Limit_l set the possible output range of Y.
the output flags lim will signal that the output limits are active and overflow will signal that the integrator has reached its limits.

since rev 1.1 the "trapezregel is used for more accuracy.
rev 1.2 added selective integratin which means the integrative component is only active within a small range of the target value 
this avoids the integrator to go to limits while an input setpoint change happened and is only causing overshoots.
the int_band is by default 100 which means the int is active all the time and if set to for example to 0.1 the integrator is only active
while the input is between 0.9 and 1.1 of the set_point value.

default values for KP = 1, TN = 1, TV = 1, LIMIT_L = -1000, LIMIT_H = +1000.
*)
IF NOT rst AND NOT manual THEN
	(* calculate the process error *)
	DIFF := dead_band(set_point - actual, Noise);
	IF ABS(diff) <= int_band AND NOT overflow THEN
		(* integrator is within int_band and needs to be run *)
		integ(in := diff, K := KI, run := TRUE, rst := FALSE, out_min := int_limit_L, out_max := int_limit_H);
		(* check if integrator has reached its limits and set overflow *)
		IF integ.Out >= int_limit_H OR integ.Out <= int_limit_L THEN overflow := TRUE; END_IF;
	ELSE
		(* int_band is exceeded, integrator needs to be cleared *)
		integ(rst := TRUE);
	END_IF;
	Y := KP * diff + integ.Out;
ELSIF rst THEN
	integ(rst := TRUE);		(* reset the integrator *)
	overflow := FALSE;		(* clear the overflow flag *)
	Y := (limit_H + Limit_L) * 0.5 - Offset;	(* set the output between limit_L and limit_L offset will be added again at the end *)
ELSIF manual THEN
	Y := manual_in;
	integ(rst := TRUE);		(* make sure integrator is reset to 0 *)
	overflow := FALSE;		(* manual operation will cancel overflow because integrator was reset *)
END_IF;

(* add offset to Y *)
Y := Y + Offset;

(* limit the outputs and set the lim flag if necessary *)
IF y > limit_H THEN
	y := limit_H;
	lim := TRUE;
ELSIF y < limit_L THEN
	y := limit_L;
	lim := TRUE;
ELSE
	lim := FALSE;
END_IF;



(* revision history
hm 	31.10.2007 	rev 1.0
	original version

hm	3.11.2007	rev 1.1
	added noise input to filter noise
	added output diff
	set limit output false when output is within limits
	overfolw was not set correctly

hm	5. jan 2008	rev 1.2
	improved performance
*)
END_FUNCTION_BLOCK

(* POU Engineering/control/FT_PID, ST *)
FUNCTION_BLOCK FT_PID
VAR_INPUT
	actual, set_point, noise, offset, manual_in : REAL;
	Manual : BOOL;
	rst : BOOL := FALSE;
	int_band : REAL := 100;
	KP : REAL := 1.0;
	TN : REAL := 1.0;
	TV : REAL := 1.0;
	limit_L : REAL := -1000;
	limit_H : REAL := 1000;
END_VAR
VAR_INPUT CONSTANT
	int_limit_L : REAL := -1000;
	int_limit_H : REAL := 1000;
END_VAR
VAR_OUTPUT
	Y : REAL;
	diff: REAL;
	LIM, overflow : BOOL;
END_VAR
VAR
	integ : FT_INT;
	deriv : FT_deriv;
END_VAR

(*
version 1.6	5 jan 2008
programmer 	hugo
tested by		tobias

FT_PID is a pid controller with manual functionality.
The PID controller works according to the fomula Y = KP * ( e + 1/TN * INTEG(e) + TV *DERIV(e)) + offset, while e = set_point - actual.
a rst will reset all internal data, while a switch to manual will cause the controller to follow the function Y = manual_in + offset.
limit_h and Limit_l set the possible output range of Y.
the output flags lim will signal that the output limits are active and overflow will signal that the integrator has reached the max or min limit.  

since rev 1.1 the "trapezregel is used for more accuracy.
rev 1.2 added selective integratin which means the integrative component is only active within a small range of the target value 
this avoids the integrator to go to limits while an input setpoint change happened and is only causing overshoots.
the int_band is by default 100 which means the int is active all the time and if set to for example to 0.1 the integrator is only active
while the input is between 0.9 and 1.1 of the set_point value.

default values for KP = 1, TN = 1, TV = 1, LIMIT_L = -1000, LIMIT_H = +1000.
*)
IF NOT rst AND NOT manual THEN
	(* calculate the process error *)
	DIFF := DEAD_BAND(set_point - actual, Noise);
	IF ABS(diff) <= int_band AND NOT overflow AND TN > 0 THEN
		(* integrator is within int_band and needs to be run *)
		integ(in := diff, K := 1/TN, run := TRUE, rst := FALSE, out_min := int_limit_L, out_max := int_limit_H);
		(* check if integrator has reached its limits and set overflow *)
		IF integ.Out >= int_limit_H OR integ.Out <= int_limit_L THEN overflow := TRUE; END_IF;
	ELSE
		(* int_band is exceeded, integrator needs to be cleared *)
		integ(rst := TRUE);
	END_IF;
	(* calculate the derivative part *)
	deriv(in := diff, K := TV);
	(* add up all parts *)
	Y := KP * (integ.Out + deriv.out + diff);
ELSIF rst THEN
	integ(rst := TRUE);		(* reset the integrator *)
	overflow := FALSE;		(* clear the overflow flag *)
	Y := (limit_H + Limit_L) * 0.5 - Offset;	(* set the output between limit_L and limit_L offset will be added again at the end *)
ELSIF manual THEN
	Y := manual_in;
	integ(rst := TRUE);		(* make sure integrator is reset to 0 *)
	overflow := FALSE;		(* manual operation will cancel overflow because integrator was reset *)
END_IF;

(* add offset to Y *)
Y := Y + Offset;

(* limit the outputs and set the lim flag if necessary *)
IF y > limit_H THEN
	y := limit_H;
	lim := TRUE;
ELSIF y < limit_L THEN
	y := limit_L;
	lim := TRUE;
ELSE
	lim := FALSE;
END_IF;


(* old code before rev 1.4
IF rst OR KP = 0 THEN
	y := Offset;
	integ(rst := 1);
	integ.rst := 0;
ELSIF manual THEN
	Y := manual_in + Offset;
	integ(rst := 1);
	integ.rst := 0;
ELSE
	(* calcualtion of the actual PID values *)
	diff := set_point - actual;

	(* integrator is only called if TN > 0 and input is within int_band othewrwise it is disabled *)
	IF TN > 0 AND actual > set_point - int_band AND actual < set_point + int_band THEN
		integ(in := diff, K := 1/TN, out_min := (limit_L - offset) / KP, out_max := (limit_H - offset) / KP);
	ELSE
		integ(rst := 1);
		integ.rst := 0;
	END_IF;
	deriv(in := diff, K := TV);

	(* check if integrator has reached the allowed limits and set overflow if necessary *)
	IF integ.Out >= (limit_H - offset) / KP THEN
		Y := limit_H;
		overflow := TRUE;
	ELSIF integ.Out <= (limit_L - offset) / KP THEN
		Y := limit_L;
		overflow := TRUE;
	ELSE
		Y := KP * (integ.Out + deriv.out + diff) + offset;
		overflow := FALSE;
	END_IF;

	(* this portion limits the output to limit_H and limit_L and set the lim flag if limits are exceeded *)
	IF Y > limit_H THEN
		Y := limit_H;
		Lim := TRUE;
	ELSIF Y < limit_L THEN
		Y := limit_L;
		lim := TRUE;
	ELSE
		lim := FALSE;
	END_IF;
END_IF;
*)

(* revision history

hm 1.12.2006	 	rev 1.1
	changed algorithm to trapezregel for higher accuracy.

hm 3.1.2007		rev 1.2
	added integ_band to select when the integrator is active.

hm	3.3.2007		rev 1.3
	added default values to inputs KP, TN, TV, LIMIT_L und LIMIT_H.

hm 31.oct 2007	rev 1.4
	total rewrite of the module to avoid failures when one of the limits is 0

hm	3.11.2007	rev 1.5
	added noise input to filter noise
	added output diff
	set limit output false when output is within limits
	overfolw was not set correctly

hm	5. jan 2008	rev 1.6
	improved code for better performance
*)
END_FUNCTION_BLOCK

(* POU Engineering/control/FT_PT2, ST *)
FUNCTION_BLOCK FT_PT2
VAR_INPUT
	in : REAL;
	T : TIME;
	D : REAL;
	K : REAL := 1;
END_VAR
VAR_OUTPUT
	out : REAL;
END_VAR
VAR
	init: BOOL;
	int1 : FT_INT;
	int2 : FT_INT;
	tn: REAL;
END_VAR

(*
version 1.3	30 Nov 2007
programmer 	hugo
tested by		tobias

FT_PT2 is a 2nd grade filter with programmable times T, D and faktor K.
 
*)
(* startup initialisation *)
IF NOT init THEN
	out := K * in;
	init := TRUE;
ELSIF T = t#0s THEN
	out := K * in;
ELSE
	tn := TIME_TO_REAL(T)/1000;
	int1(in := in * K / (TN * TN) - int1.Out * 2 *D / TN - int2.Out / (TN * TN));
	int2(in := int1.Out);
	out := int2.out;
END_IF;

(* revision history

15.1.2007 hm		rev 1.1
	changed formula to new more acurate formula
	old code:
	tx := TIME();
	IF NOT init THEN
		last := tx;
		init := TRUE;
	ELSE
		IF T> t#0s THEN
			out1 := out1 + (in - out1) * TIME_TO_REAL(Tx - last) / TIME_TO_REAL(T);
		ELSE
			out1 := in;
		END_IF;
		IF T > t#0s THEN
			out2 := out2 + (out1 - out2) * TIME_TO_REAL(Tx - last) / TIME_TO_REAL(T);
		ELSE
			out2 := out1;
		END_IF;
		out := out2 * K;
	END_IF;
	last := tx;

hm 		15.9.2007		rev 1.2
	deleted unused code for init system time reading tx	

hm		30.11.2007		rev 1.3
	changed out to be K * in during initialization
	avoind divide by 0 if tn = 0
*)
END_FUNCTION_BLOCK

(* POU Engineering/control/FT_TN16, ST *)
FUNCTION_BLOCK FT_TN16
VAR_INPUT
	in : REAL;
	T : TIME;
END_VAR
VAR_OUTPUT
	out : REAL;
	trig : BOOL;
END_VAR
VAR
	length : INT := 16;
	X : ARRAY[0..15] OF REAL;
	cnt : INT;
	last : TIME;
	tx: TIME;
	init: BOOL;
END_VAR

(*
version 1.1	16 sep 2007
programmer 	hugo
tested by		tobias

FT_TN16 is delay function, it will delay a signal by a specified time : T and will store 16 values of in before they are put thru to out.
for higher or lower resolution please use FT_TN8 or FT_TN64 instead.
 
*)
(* read system time *)
tx := DWORD_TO_TIME(T_PLC_MS());

trig := FALSE;
IF NOT init THEN
	x[cnt] := in;
	init := TRUE;
	last := tx;
ELSIF tx - last >= T / length THEN
	IF cnt = length - 1 THEN cnt := 0; ELSE cnt := cnt + 1; END_IF;
	Out := X[cnt];
	x[cnt] := in;
	last := tx;
	Trig := TRUE;
END_IF;

(* revision history
hm		1. jan 2007		rev 1.0
	original version

hm		16. sep 2007	rev 1.1
	changes time() to T_plc_ms() for compatibility reasons

*)
END_FUNCTION_BLOCK

(* POU Engineering/control/FT_TN64, ST *)
FUNCTION_BLOCK FT_TN64
VAR_INPUT
	in : REAL;
	T : TIME;
END_VAR
VAR_OUTPUT
	out : REAL;
	trig: BOOL;
END_VAR
VAR
	length : INT := 64;
	X : ARRAY[0..63] OF REAL;
	cnt : INT;
	last : TIME;
	tx: TIME;
	init: BOOL;
END_VAR

(*
version 1.1	15 sep 2007
programmer 	hugo
tested by		tobias

FT_TN7 is delay function, it will delay a signal by a specified time : T and will store 64 values of in before they are put thru to out.
if lower resolution is needed, pls use FT_TN8 or FT_TN16 instead.
 
*)
(* read system time *)
tx := DWORD_TO_TIME(T_PLC_MS());

trig := FALSE;
IF NOT init THEN
	x[cnt] := in;
	init := TRUE;
	last := tx;
ELSIF tx - last >= T / length THEN
	IF cnt = length - 1 THEN cnt := 0; ELSE cnt := cnt + 1; END_IF;
	Out := X[cnt];
	x[cnt] := in;
	last := tx;
	trig := TRUE;
END_IF;

(* revision history
hm		1. jan 2007		rev 1.0
	original version

hm		16. sep 2007	rev 1.1
	changes time() to T_plc_ms() for compatibility reasons

*)
END_FUNCTION_BLOCK

(* POU Engineering/control/FT_TN8, ST *)
FUNCTION_BLOCK FT_TN8
VAR_INPUT
	in : REAL;
	T : TIME;
END_VAR
VAR_OUTPUT
	out : REAL;
	trig: BOOL;
END_VAR
VAR
	length : INT := 8;
	X : ARRAY[0..7] OF REAL;
	cnt : INT;
	last : TIME;
	tx: TIME;
	init: BOOL;
END_VAR

(*
version 1.1	15 Sep 2007
programmer 	hugo
tested by		tobias

FT_TN8 is delay function, it will delay a signal by a specified time : T and will store 8 values of in before they are put thru to out.
if higher resolution is needed, pls use FT_TN16 or FT_TN64 instead.
 
*)
tx := DWORD_TO_TIME(T_PLC_MS());
trig := FALSE;
IF NOT init THEN
	x[cnt] := in;
	init := TRUE;
	last := tx;
ELSIF tx - last >= T / length THEN
	IF cnt = length - 1 THEN cnt := 0; ELSE cnt := cnt + 1; END_IF;
	Out := X[cnt];
	x[cnt] := in;
	last := tx;
	trig := TRUE;
END_IF;

(* revision history
hm		1. jan 2007		rev 1.0
	original version

hm		16. sep 2007	rev 1.1
	changes time() to T_plc_ms() for compatibility reasons

*)
END_FUNCTION_BLOCK

(* POU Engineering/control/hyst_2, ST *)
FUNCTION_BLOCK hyst_2
VAR_INPUT
	In : REAL;
	val : REAL;
	hys : REAL;
END_VAR
VAR_OUTPUT
	Q : BOOL := 0;
	win: BOOL;
END_VAR
VAR
	X : REAL;
END_VAR


(*
	version 1.1	5. jan 2008
	programmer 	oscat
	tested BY		tobias

this hysteresis function switches the output high if the input signal reaches obove val + hys/2 and will switch to low when the input falls back below val - hys/2 value.
a separate output mid is set if the input stays between low and high value.

*)
X := hys * 0.5;
IF Q THEN
	IF in < val - x THEN q := FALSE; END_IF;
ELSE
	IF in > val + x THEN q := TRUE; END_IF;
END_IF;
win := in > val - x AND in < val + x;


(* revision history
hm	4. aug 2006		rev 1.0
	original version

hm	5. jan 2008		rev 1.1
	improved code for better performance

*)
END_FUNCTION_BLOCK

(* POU Engineering/control/Hyst_3, ST *)
FUNCTION_BLOCK Hyst_3
VAR_INPUT
	in : REAL;
	hyst : REAL;
	val1 : REAL;
	val2 : REAL;
END_VAR
VAR_OUTPUT
	Q1 : BOOL;
	Q2 : BOOL;
END_VAR
VAR
	X: REAL;
END_VAR

(*
	version 1.2	5 jan 2008
	programmer 	oscat
	tested BY		tobias

this is a double hysteresis function. Out1 follows a hysteresis function defined by val1and hyst, while out 2 follows val2 and hyst.
if the input signal is between the two hysteresis switches (val1 and val2) then non of the outputs is active.

*)
X := hyst * 0.5;
IF in < val1 - X THEN
	q1 := TRUE;
ELSIF in > val1 + X THEN
	q1 := FALSE;
END_IF;
IF in < val2 - X THEN
	q2 := FALSE;
ELSIF in > val2 + X THEN
	q2 := TRUE;
END_IF;

(* revision history
hm	22. jan 2007	rev 1.0
	original version

hm	27. dec 2007	rev 1.1
	changed code for better performance

hm	5. jan 2008		rev 1.2
	further performance iprovements

*)
END_FUNCTION_BLOCK

(* POU Engineering/conversion/astro, ST *)
FUNCTION_BLOCK astro
VAR_INPUT
	m : REAL;
	AE : REAL;
	PC : REAL;
	LJ : REAL;
END_VAR
VAR_OUTPUT
	Ym : REAL;
	YAE : REAL;
	YPC : REAL;
	YLJ : REAL;
END_VAR
VAR
END_VAR

(*
version 1.0	27 mar 2007
programmer 	hugo
tested by		oscat

this function converts different length units
any unused input can simply be left open.
different inputs connected at the same time will be added up.

*)
YAE :=	AE
		+ m / 149.597870E9
		+ PC * 206265
		+ LJ * 63240;
Ym := YAE * 149.597870E9;
YPC := YAE / 206265;
YLJ := YAE / 63240;


(*
Länge Meter m SI-Basiseinheit
Astronomische Einheit* AE 1 AE = 149,597 870 · E9 m
Parsec pc 1 pc = 206265 AE = 30,857 · E15 m
Lichtjahr Lj 1 Lj = 9,460 530 · E15 m = 63240 AE = 0,306 59 pc
Ångström Å 1 Å = E–l0 m
typograph. Punkt p 1 p = 0,376 065 mm • im Druckereigewerbe
inch** in 1 in = 2,54 · E–2 m = 25,4 mm***
foot ft 1 ft = 0,3048 m = 30,48 cm
yard yd 1 yd = 0,9144 m
mile mile 1 mile = 1609,344 m
Internat. Seemeile sm 1 sm = 1852 m
Fathom fm 1 fm = 1,829 m • in der Seeschifffahrt

*)
END_FUNCTION_BLOCK

(* POU Engineering/conversion/C_to_K, ST *)
FUNCTION C_to_K : REAL
VAR_INPUT
	Celsius : REAL;
END_VAR
VAR
END_VAR

(*
version 1.0	4 dec 2006
programmer 	hugo
tested by		tobias

this function converts celsius to kelvin
*)
C_to_K := Celsius - 273.15;
END_FUNCTION

(* POU Engineering/conversion/energy, ST *)
FUNCTION_BLOCK energy
VAR_INPUT
	J : REAL;
	C : REAL;
	Wh : REAL;
END_VAR
VAR_OUTPUT
	YJ : REAL;
	YC : REAL;
	YWh : REAL;
END_VAR
VAR
END_VAR

(*
version 1.0	27 mar 2007
programmer 	hugo
tested by		oscat

this function converts different energy units
any unused input can simply be left open.
different inputs connected at the same time will be added up.
*)
YJ := J + Wh * 3600 + C * 4.1868;
YC := YJ / 4.1868;
YWh := YJ / 3600;

(*
Arbeit, Energie, Joule* J 1 J = 1 N · m = 1 W · s = (1/3,6) E–6 kW · h = 1 kg · m2/s2
Wärmemenge Kilowattstunde kW · h 1 kW · h = 3,6 MJ = 860 kcal
Elektronvolt eV 1 eV = 160,218 92 E–21 J
Erg erg 1 erg = 1E–7 J
Kalorie cal 1 cal = 4,1868 J = 1,163 E–3 W · h
Therm therm 1 therm = 105,50 · 106 J

*)
END_FUNCTION_BLOCK

(* POU Engineering/conversion/F_to_OM, ST *)
FUNCTION F_to_OM : REAL
VAR_INPUT
	F : REAL;
END_VAR
VAR
END_VAR

(*
version 1.0	22 jan 2007
programmer 	hugo
tested by		tobias

this function converts frequency to Omega F
Omega = 2*PI*F
*)
F_to_OM := PI2 * F;
END_FUNCTION

(* POU Engineering/conversion/F_to_PT, ST *)
FUNCTION F_to_PT : TIME
VAR_INPUT
	F : REAL;
END_VAR
VAR
END_VAR

(*
version 1.0	4 aug 2006
programmer 	hugo
tested by		tobias

this function converts frequency to periode time  
*)
F_to_PT := DWORD_TO_TIME(REAL_TO_DWORD(1/F*1000));
END_FUNCTION

(* POU Engineering/conversion/K_to_C, ST *)
FUNCTION K_to_C : REAL
VAR_INPUT
	Kelvin : REAL;
END_VAR
VAR
END_VAR

(*
version 1.0	4 dec 2006
programmer 	hugo
tested by		tobias

this function converts kelvin to celsius
*)
K_to_C := Kelvin + 273.15;
END_FUNCTION

(* POU Engineering/conversion/KMH_TO_MS, ST *)
FUNCTION KMH_TO_MS : REAL
VAR_INPUT
	kmh : REAL;
END_VAR
VAR
END_VAR

(*
version 1.1	6 jan 2007
programmer 	hugo
tested by		tobias

this function converts velocities from Kilometers / hour to Meters / Second

*)
KMH_TO_MS := kmh * 0.2777777777777;

(* revision history
hm	4. feb 2007		rev 1.0
	original version

hm	6. jan 2008		rev 1.1
	improved performance

*)
END_FUNCTION

(* POU Engineering/conversion/MS_TO_KMH, ST *)
FUNCTION MS_TO_KMH : REAL
VAR_INPUT
	ms : REAL;
END_VAR
VAR
END_VAR

(*
version 1.0	4 Feb 2007
programmer 	hugo
tested by		tobias

this function converts velocities from Meters / Second to Kilometers / hour.

*)
MS_TO_KMH := ms * 3.6;
END_FUNCTION

(* POU Engineering/conversion/OM_to_F, ST *)
FUNCTION OM_to_F : REAL
VAR_INPUT
	OM : REAL;
END_VAR
VAR
END_VAR

(*
version 1.0	22 jan 2007
programmer 	hugo
tested by		tobias

this function converts Omega F to frequency
F = OM / (2*PI)
*)
OM_to_F := OM / PI2;
END_FUNCTION

(* POU Engineering/conversion/PT_to_F, ST *)
FUNCTION PT_to_F : REAL
VAR_INPUT
	PT : TIME;
END_VAR
VAR
END_VAR

(*
version 1.0	4 aug 2006
programmer 	hugo
tested by		tobias

this function converts periode time to frequency
*)
PT_to_F := 1000/DWORD_TO_REAL(TIME_TO_DWORD(PT));
END_FUNCTION

(* POU Engineering/conversion/Temperature, ST *)
FUNCTION_BLOCK Temperature
VAR_INPUT
	K : REAL;
	C : REAL := -273.15;
	F : REAL := -459.67;
	Re : REAL := -218.52;
	Ra : REAL := 0;
END_VAR
VAR_OUTPUT
	YK : REAL;
	YC : REAL;
	YF : REAL;
	YRe : REAL;
	YRa : REAL;
END_VAR
VAR
END_VAR

(*
version 1.0	21 feb 2008
programmer 	hugo
tested by	oscat

this function converts different temperature units
any unused input can simply be left open.
different inputs connected at the same time will be added up.

*)
YK := K + (C + 273.15) + (F + 459.67) * 0.555555555555 + (Re * 1.25 + 273.15) + (Ra * 0.555555555555);
YC := YK -273.15;
YF := YK * 1.8 - 459.67;
YRe := (YK - 273.15) * 0.8;
YRa := YK * 1.8;


(* revision history
hm	21. feb. 2008	rev 1.0
	original version

*)
END_FUNCTION_BLOCK

(* POU Engineering/measurements/bar_graph, ST *)
FUNCTION_BLOCK bar_graph
VAR_INPUT
	X : REAL;
	rst : BOOL;
END_VAR
VAR_INPUT CONSTANT
	trigger_Low : REAL;
	trigger_High : REAL;
	Alarm_low : BOOL;
	Alarm_high : BOOL;
	log_scale : BOOL;
END_VAR
VAR_OUTPUT
	LOW, Q1, Q2, Q3, Q4, Q5, Q6, HIGH : BOOL;
	Alarm : BOOL;
	Status : BYTE;
END_VAR
VAR
	init : BOOL;
	T1, T2, T3, T4, T5 : REAL;
END_VAR
VAR_TEMP
	temp : REAL;
END_VAR

(*
	version 1.2	6 jan 2008
	programmer 	hugo
	tested BY		hans

bar graph is a muti window comparator which displays an analog input signal on 8 digital outputs.
only one output is active a any given time depending on the value of the input signal.
the output can be of linear or logarithmic scale.

*)
IF NOT init THEN
	init := TRUE;
	IF log_scale THEN
		temp := EXP(LN(Trigger_high / Trigger_low) * 0.166666666666666666666);
		T1 := trigger_low * temp;
		T2 := T1 * temp;
		T3 := T2 * temp;
		T4 := T3 * temp;
		T5 := T4 * temp;
	ELSE
		temp := (trigger_high - trigger_low) * 0.142857142;
		T1 := trigger_low + temp;
		T2 := T1 + temp;
		T3 := T2 + temp;
		T4 := T3 + temp;
		T5 := T4 + temp;
	END_IF;
END_IF;

(* clear outputs before checking *)
Q1 := FALSE;
Q2 := FALSE;
Q3 := FALSE;
Q4 := FALSE;
Q5 := FALSE;
Q6 := FALSE;
status := 110;

(* low, high and alarm can only be cleared with rst depending on alarm_low and alarm_high *)
IF NOT alarm_low THEN low := FALSE; END_IF;
IF NOT alarm_high THEN high := FALSE; END_IF;
IF rst THEN
	alarm := FALSE;
	low := FALSE;
	high := FALSE;
END_IF;

(* check and set outputs *)
IF X < trigger_low THEN
	Low := TRUE;
	status := 111;
	IF alarm_low THEN
		alarm := TRUE;
		status := 1;
	END_IF;
ELSIF X < T1 THEN
	Q1 := TRUE;
ELSIF x < t2 THEN
	Q2 := TRUE;
ELSIF x < t3 THEN
	Q3 := TRUE;
ELSIF x < T4 THEN
	Q4 := TRUE;
ELSIF x < T5 THEN
	q5 := TRUE;
ELSIF x < trigger_high THEN
	q6 := TRUE;
ELSE
	high := TRUE;
	status := 112;
	IF alarm_high THEN
		alarm := TRUE;
		status := 2;
	END_IF;
END_IF;

(* revision history
hm	22. feb 2007	rev 1.0
	original version

hm	2. dec 2007		rev 1.1
	chaged code for better performance

hm	6. jan 2008		rev 1.2
	further performance improvement

*)
END_FUNCTION_BLOCK

(* POU Engineering/measurements/Calibrate, ST *)
FUNCTION_BLOCK Calibrate
VAR_INPUT
	X : REAL;
	CO : BOOL;
	CS : BOOL;
END_VAR
VAR_INPUT CONSTANT
	Y_Offset : REAL;
	Y_Scale : REAL;
END_VAR
VAR_OUTPUT
	Y : REAL;
END_VAR
VAR RETAIN
	offset : REAL;
	Scale : REAL := 1;
END_VAR

(*
	version 1.2	22 feb 2007
	programmer 	hugo
	tested BY		hans

Calibrate allows for offset and scale calibration of an analog input.
offset is calibrated to a stored reference Y_offset while CO is true.
after the offset is calibrated, scale can be calibrated to a reference value Y_scale while CS is true.
*)
(* check for calibration *)
IF CO THEN
	Offset := Y_Offset - X;
ELSIF CS THEN
	scale := Y_scale / (X+Offset);
END_IF;
(* calculate output *)
Y := (X + Offset) * Scale;


(* revision history
hm 22.2.2007		rev 1.2
	changed VAR RETAIN PERSISTENT to VAR RETAIN for better compatibility
	wago lon contollers do not support persisitent

*)
END_FUNCTION_BLOCK

(* POU Engineering/measurements/m_d, ST *)
FUNCTION_BLOCK m_d
VAR_INPUT
	start : BOOL;
	stop : BOOL;
	tmax : TIME := t#10d;
	rst: BOOL;
END_VAR
VAR_OUTPUT
	PT : TIME := t#0ms;
	ET : TIME;
	run : BOOL;
END_VAR
VAR
	edge : BOOL := 0;
	T0 : TIME;
	tx: TIME;
	startup: BOOL;
END_VAR

(*
	version 1.1	16 sep 2007
	programmer 	hugo
	tested BY		tobias

m_d measures the time between a rising edge on start to a rising edge on stop and returs the last measured value on the output PT.
a second output ET is starting from 0 at the rising edge of start and is counting up until the rising edge of stop occurs.
the asynchronous input rst can reset the outputs at any time.
tmax defines a timeout wich is the maximum measurable time between start and stop, if this time is exceeded the outputs will stay at 0.
*)
(* check for rst input *)
IF rst OR et >= tmax THEN
	pt := t#0ms;
	et := t#0ms;
	startup := FALSE;
	run := FALSE;
END_IF;

(* avoid timers to start when input is true at startup *)
IF NOT startup THEN
	edge := start;
	startup := TRUE;
END_IF;

(* read system timer *)
tx := DWORD_TO_TIME(T_PLC_MS());

(* detect rising edge on start *)
IF start AND NOT edge AND NOT stop THEN
	t0 := tx;
	run := TRUE;
	pt := t#0s;
ELSIF stop AND run THEN
	pt := et;
	run := FALSE;
END_IF;
edge := start;
IF run THEN et := tx - t0; END_IF;

(* revision history
hm		2.5.2007	rev 1.0
	original version

hm		16.9.2007	rev 1.1
	changes time() to T_plc_ms() for compatibility reasons

*)
END_FUNCTION_BLOCK

(* POU Engineering/measurements/m_t, ST *)
FUNCTION_BLOCK m_t
VAR_INPUT
	in: BOOL;
	tmax : TIME := t#10d;
	rst: BOOL;
END_VAR
VAR_OUTPUT
	PT : TIME := t#0ms;
	ET: TIME;
END_VAR
VAR
	edge : BOOL := 0;
	start : TIME;
	stop : TIME;
	init : BOOL;
	tx: TIME;
	startup: BOOL;
END_VAR

(*
	version 1.2	16 sep 2007
	programmer 	hugo
	tested BY		tobias

m_t measures the with of a high pulse and returs the last measured pulse width on output PT.
a second output ET is starting from 0 at the rising edge and counting up until the falling edge occurs and resetts et to 0.
the asynchrtonous input rst can reset the outputs at any time.
tmax defines a maximum measurable time, if this value is exceeded the outputs will be reset to 0.
*)
(* check for rst input *)
IF rst OR et >= tmax THEN
	init := FALSE;
	startup := FALSE;
	pt := t#0ms;
	et := t#0ms;
END_IF;

(* avoid timers to start when input is true at startup *)
IF NOT startup THEN
	edge := in;
	startup := TRUE;
END_IF;

(* read system timer *)
tx := DWORD_TO_TIME(T_PLC_MS());

(* edge trigger rising and falling edge *)
IF in XOR edge THEN
	edge := in;
	(* rising edge starts measurement *)
	IF in THEN
		init := TRUE;
		start := Tx;
	(* falling edge stops measurement *)
	ELSIF init THEN
		stop := Tx;
		pt := stop - start;
	END_IF;
END_IF;

IF init AND in THEN
	et := Tx - start; ELSE et := t#0ms;
END_IF;

(* revision history
hm		4.8.2006	rev 1.0
	original version

hm		2.5.2007	rev 1.1
	added init variable to avoid unreasonable measurement if falling edge occurs first.
	added et (elapsed time) output to count from 0 at rising edge until a falling edge resets et to 0.
	added reset input.

hm		16.9.2007	rev 1.2
	changes time() to T_plc_ms() for compatibility reasons

*)
END_FUNCTION_BLOCK

